KUKA KRL program: f1_Kuka_APT218T03S18.SRC

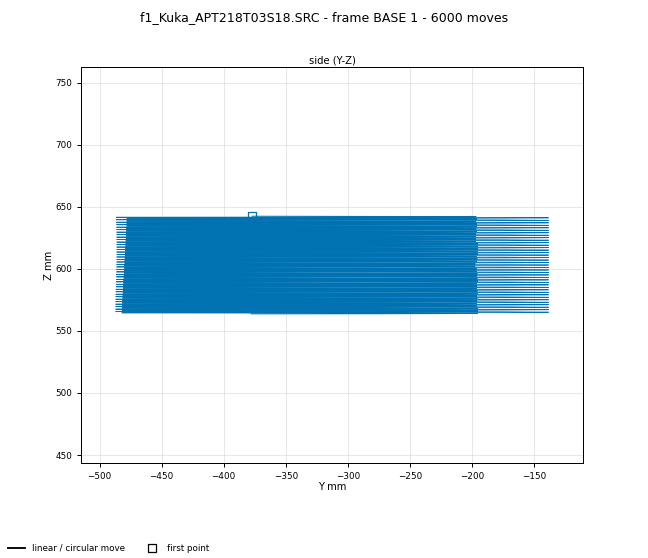
[picture p0: tool path of f1_Kuka_APT218T03S18.SRC in frame BASE 1, 6000 of 6001 moves have a stored position in this frame; points joined in program order, loops and branches not executed]
&ACCESS RVP
&REL 2
&PARAM TEMPLATE = C:\KRC\Roboter\Template\vorgabe
&PARAM EDITMASK = *
DEF f1_Kuka_APT218T03S18()


;FOLD INI;%{PE}%V3.2.0,%MKUKATPBASIS,%CINIT,%VCOMMON,%P
  ;FOLD BAS INI;%{E}%V3.2.0,%MKUKATPBASIS,%CINIT,%VINIT,%P
    GLOBAL INTERRUPT DECL 3 WHEN $STOPMESS==TRUE DO IR_STOPM ( )
    INTERRUPT ON 3
    BAS (#INITMOV,0 )
  ;ENDFOLD (BAS INI)
  ;FOLD USER INI;%{E}%V3.2.0,%MKUKATPUSER,%CINIT,%VINIT,%P
    ;Make your modifications here
  ;ENDFOLD (USER INI)
;ENDFOLD (INI)


;*** Make Null PTP Move
  PTP $pos_act

;*** Auto Load The Correct TOOL Data
  $tool=tool_data[3]

;*** Auto Load The Correct BASE Data
  $base=base_data[1]

  $ADVANCE = 5

;*** Restate Last Velocity
MMPM(30000.0)
SetRPM(6000)
LIN {X -0.101,Y -377.217,Z 642.442,A 0.000,B 0.000,C 90.000,E1 79.634} C_DIS
LIN {X 0.001,Y -366.007,Z 642.429,A 0.000,B 0.000,C 90.000,E1 77.285} C_DIS
LIN {X 0.196,Y -351.281,Z 642.411,A 0.000,B 0.000,C 90.000,E1 73.976} C_DIS
LIN {X -0.048,Y -341.253,Z 642.398,A 0.000,B 0.000,C 90.000,E1 71.583} C_DIS
LIN {X 0.012,Y -327.143,Z 642.377,A 0.000,B 0.000,C 90.000,E1 67.847} C_DIS
LIN {X 0.084,Y -314.471,Z 642.356,A 0.000,B 0.000,C 90.000,E1 64.024} C_DIS
LIN {X 0.048,Y -304.930,Z 642.338,A 0.000,B 0.000,C 90.000,E1 60.795} C_DIS
LIN {X -0.099,Y -296.125,Z 642.320,A 0.000,B 0.000,C 90.000,E1 57.533} C_DIS
LIN {X -0.021,Y -289.495,Z 642.305,A 0.000,B 0.000,C 90.000,E1 54.848} C_DIS
LIN {X -0.014,Y -283.083,Z 642.290,A 0.000,B 0.000,C 90.000,E1 52.145} C_DIS
LIN {X 0.119,Y -278.142,Z 642.278,A 0.000,B 0.000,C 90.000,E1 50.070} C_DIS
LIN {X 0.131,Y -272.810,Z 642.267,A 0.000,B 0.000,C 90.000,E1 48.000} C_DIS
LIN {X -0.152,Y -266.946,Z 642.255,A 0.000,B 0.000,C 90.000,E1 45.972} C_DIS
LIN {X -0.168,Y -260.527,Z 642.243,A 0.000,B 0.000,C 90.000,E1 43.866} C_DIS
LIN {X 0.065,Y -253.879,Z 642.232,A 0.000,B 0.000,C 90.000,E1 41.676} C_DIS
LIN {X -0.149,Y -243.020,Z 642.211,A 0.000,B 0.000,C 90.000,E1 38.096} C_DIS
LIN {X -0.001,Y -234.963,Z 642.195,A 0.000,B 0.000,C 90.000,E1 35.105} C_DIS
LIN {X 0.062,Y -227.705,Z 642.178,A 0.000,B 0.000,C 90.000,E1 32.084} C_DIS
LIN {X -0.103,Y -221.117,Z 642.161,A 0.000,B 0.000,C 90.000,E1 29.077} C_DIS
LIN {X -0.063,Y -215.336,Z 642.144,A 0.000,B 0.000,C 90.000,E1 25.976} C_DIS
LIN {X 0.066,Y -209.174,Z 642.122,A 0.000,B 0.000,C 90.000,E1 22.025} C_DIS
LIN {X 0.077,Y -204.198,Z 642.100,A 0.000,B 0.000,C 90.000,E1 18.055} C_DIS
LIN {X 0.016,Y -200.306,Z 642.078,A 0.000,B 0.000,C 90.000,E1 14.064} C_DIS
LIN {X 0.027,Y -196.658,Z 642.047,A 0.000,B 0.000,C 90.000,E1 8.398} C_DIS
LIN {X -0.004,Y -197.458,Z 641.952,A 0.000,B 0.000,C 90.000,E1 351.376} C_DIS
LIN {X -0.032,Y -200.895,Z 641.925,A 0.000,B 0.000,C 90.000,E1 346.520} C_DIS
LIN {X -0.002,Y -204.863,Z 641.903,A 0.000,B 0.000,C 90.000,E1 342.489} C_DIS
LIN {X -0.060,Y -209.769,Z 641.881,A 0.000,B 0.000,C 90.000,E1 338.518} C_DIS
LIN {X 0.082,Y -215.497,Z 641.859,A 0.000,B 0.000,C 90.000,E1 334.537} C_DIS
LIN {X -0.009,Y -221.886,Z 641.837,A 0.000,B 0.000,C 90.000,E1 330.667} C_DIS
LIN {X 0.024,Y -227.475,Z 641.820,A 0.000,B 0.000,C 90.000,E1 327.582} C_DIS
LIN {X 0.036,Y -234.865,Z 641.799,A 0.000,B 0.000,C 90.000,E1 323.783} C_DIS
LIN {X -0.064,Y -242.913,Z 641.778,A 0.000,B 0.000,C 90.000,E1 320.070} C_DIS
LIN {X 0.005,Y -251.812,Z 641.758,A 0.000,B 0.000,C 90.000,E1 316.377} C_DIS
LIN {X -0.006,Y -261.731,Z 641.738,A 0.000,B 0.000,C 90.000,E1 312.771} C_DIS
LIN {X 0.117,Y -271.858,Z 641.720,A 0.000,B 0.000,C 90.000,E1 309.564} C_DIS
LIN {X 0.057,Y -283.236,Z 641.703,A 0.000,B 0.000,C 90.000,E1 306.457} C_DIS
LIN {X -0.012,Y -295.817,Z 641.686,A 0.000,B 0.000,C 90.000,E1 303.420} C_DIS
LIN {X -0.138,Y -309.656,Z 641.669,A 0.000,B 0.000,C 90.000,E1 300.463} C_DIS
LIN {X 0.023,Y -323.063,Z 641.655,A 0.000,B 0.000,C 90.000,E1 297.847} C_DIS
LIN {X -0.032,Y -335.104,Z 641.642,A 0.000,B 0.000,C 90.000,E1 295.643} C_DIS
LIN {X 0.079,Y -351.402,Z 641.627,A 0.000,B 0.000,C 90.000,E1 292.845} C_DIS
LIN {X -0.048,Y -370.901,Z 641.610,A 0.000,B 0.000,C 90.000,E1 289.866} C_DIS
LIN {X -0.020,Y -386.121,Z 641.599,A 0.000,B 0.000,C 90.000,E1 287.819} C_DIS
LIN {X -0.151,Y -402.387,Z 641.588,A 0.000,B 0.000,C 90.000,E1 285.843} C_DIS
LIN {X 0.020,Y -414.001,Z 641.580,A 0.000,B 0.000,C 90.000,E1 284.426} C_DIS
LIN {X -0.039,Y -425.082,Z 641.573,A 0.000,B 0.000,C 90.000,E1 283.063} C_DIS
LIN {X -0.027,Y -435.735,Z 641.565,A 0.000,B 0.000,C 90.000,E1 281.715} C_DIS
LIN {X -0.081,Y -443.889,Z 641.559,A 0.000,B 0.000,C 90.000,E1 280.658} C_DIS
LIN {X -0.145,Y -456.034,Z 641.550,A 0.000,B 0.000,C 90.000,E1 279.095} C_DIS
LIN {X -0.043,Y -464.453,Z 641.545,A 0.000,B 0.000,C 90.000,E1 278.049} C_DIS
LIN {X -0.153,Y -470.095,Z 641.540,A 0.000,B 0.000,C 90.000,E1 277.296} C_DIS
LIN {X 0.259,Y -474.932,Z 641.536,A 0.000,B 0.000,C 90.000,E1 276.486} C_DIS
LIN {X 0.187,Y -478.977,Z 641.532,A 0.000,B 0.000,C 90.000,E1 275.739} C_DIS
LIN {X -0.142,Y -481.189,Z 641.529,A 0.000,B 0.000,C 90.000,E1 275.277} C_DIS
LIN {X 0.019,Y -482.986,Z 641.526,A 0.000,B 0.000,C 90.000,E1 274.759} C_DIS
LIN {X 0.149,Y -484.460,Z 641.524,A 0.000,B 0.000,C 90.000,E1 274.245} C_DIS
LIN {X -0.157,Y -485.468,Z 641.521,A 0.000,B 0.000,C 90.000,E1 273.784} C_DIS
LIN {X -0.002,Y -486.133,Z 641.518,A 0.000,B 0.000,C 90.000,E1 273.269} C_DIS
LIN {X 0.187,Y -486.492,Z 641.515,A 0.000,B 0.000,C 90.000,E1 272.751} C_DIS
LIN {X -0.130,Y -486.583,Z 641.513,A 0.000,B 0.000,C 90.000,E1 272.293} C_DIS
LIN {X 0.058,Y -486.383,Z 641.510,A 0.000,B 0.000,C 90.000,E1 271.776} C_DIS
LIN {X 0.230,Y -485.845,Z 641.507,A 0.000,B 0.000,C 90.000,E1 271.260} C_DIS
LIN {X -0.083,Y -484.907,Z 641.504,A 0.000,B 0.000,C 90.000,E1 270.802} C_DIS
LIN {X 0.088,Y -483.494,Z 641.502,A 0.000,B 0.000,C 90.000,E1 270.286} C_DIS
LIN {X -0.230,Y -481.516,Z 641.499,A 0.000,B 0.000,C 90.000,E1 269.828} C_DIS
LIN {X -0.074,Y -478.834,Z 641.496,A 0.000,B 0.000,C 90.000,E1 269.312} C_DIS
LIN {X 0.061,Y -475.404,Z 641.493,A 0.000,B 0.000,C 90.000,E1 268.797} C_DIS
LIN {X 0.175,Y -470.957,Z 641.491,A 0.000,B 0.000,C 90.000,E1 268.282} C_DIS
LIN {X 0.002,Y -468.333,Z 641.489,A 0.000,B 0.000,C 90.000,E1 268.051} C_DIS
LIN {X -0.184,Y -465.346,Z 641.488,A 0.000,B 0.000,C 90.000,E1 267.822} C_DIS
LIN {X -0.130,Y -462.383,Z 641.487,A 0.000,B 0.000,C 90.000,E1 267.593} C_DIS
LIN {X -0.076,Y -459.035,Z 641.485,A 0.000,B 0.000,C 90.000,E1 267.364} C_DIS
LIN {X 0.127,Y -452.068,Z 641.483,A 0.000,B 0.000,C 90.000,E1 266.963} C_DIS
LIN {X 0.044,Y -444.600,Z 641.482,A 0.000,B 0.000,C 90.000,E1 266.674} C_DIS
LIN {X 0.025,Y -436.739,Z 641.480,A 0.000,B 0.000,C 90.000,E1 266.445} C_DIS
LIN {X 0.024,Y -427.995,Z 641.479,A 0.000,B 0.000,C 90.000,E1 266.274} C_DIS
LIN {X -0.186,Y -419.938,Z 641.479,A 0.000,B 0.000,C 90.000,E1 266.216} C_DIS
LIN {X -0.026,Y -411.170,Z 641.479,A 0.000,B 0.000,C 90.000,E1 266.159} C_DIS
LIN {X -0.034,Y -180.927,Z 641.479,A 0.000,B 0.000,C 90.000,E1 266.159} C_DIS
LIN {X 0.072,Y -180.902,Z 641.474,A 0.000,B 0.000,C 90.000,E1 265.241} C_DIS
LIN {X 0.021,Y -180.228,Z 641.464,A 0.000,B 0.000,C 90.000,E1 263.571} C_DIS
LIN {X -0.025,Y -179.041,Z 641.446,A 0.000,B 0.000,C 90.000,E1 260.208} C_DIS
LIN {X 0.037,Y -178.709,Z 641.441,A 0.000,B 0.000,C 90.000,E1 259.342} C_DIS
LIN {X -0.069,Y -175.758,Z 641.413,A 0.000,B 0.000,C 90.000,E1 254.283} C_DIS
LIN {X -0.019,Y -171.942,Z 641.384,A 0.000,B 0.000,C 90.000,E1 249.135} C_DIS
LIN {X -0.044,Y -171.326,Z 641.379,A 0.000,B 0.000,C 90.000,E1 248.284} C_DIS
LIN {X 0.010,Y -167.582,Z 641.355,A 0.000,B 0.000,C 90.000,E1 243.948} C_DIS
LIN {X -0.052,Y -166.217,Z 641.346,A 0.000,B 0.000,C 90.000,E1 242.231} C_DIS
LIN {X -0.063,Y -162.980,Z 641.326,A 0.000,B 0.000,C 90.000,E1 238.742} C_DIS
LIN {X -0.015,Y -160.894,Z 641.312,A 0.000,B 0.000,C 90.000,E1 236.087} C_DIS
LIN {X -0.038,Y -157.663,Z 641.292,A 0.000,B 0.000,C 90.000,E1 232.557} C_DIS
LIN {X -0.099,Y -155.701,Z 641.277,A 0.000,B 0.000,C 90.000,E1 229.908} C_DIS
LIN {X -0.044,Y -151.964,Z 641.252,A 0.000,B 0.000,C 90.000,E1 225.405} C_DIS
LIN {X -0.027,Y -150.205,Z 641.237,A 0.000,B 0.000,C 90.000,E1 222.690} C_DIS
LIN {X -0.012,Y -146.973,Z 641.212,A 0.000,B 0.000,C 90.000,E1 218.141} C_DIS
LIN {X 0.007,Y -145.560,Z 641.197,A 0.000,B 0.000,C 90.000,E1 215.391} C_DIS
LIN {X 0.006,Y -142.952,Z 641.171,A 0.000,B 0.000,C 90.000,E1 210.797} C_DIS
LIN {X -0.063,Y -141.577,Z 641.151,A 0.000,B 0.000,C 90.000,E1 207.129} C_DIS
LIN {X -0.016,Y -139.415,Z 641.114,A 0.000,B 0.000,C 90.000,E1 200.610} C_DIS
LIN {X 0.037,Y -139.139,Z 641.104,A 0.000,B 0.000,C 90.000,E1 198.725} C_DIS
LIN {X 0.063,Y -138.348,Z 641.057,A 0.000,B 0.000,C 90.000,E1 190.310} C_DIS
LIN {X 0.051,Y -139.493,Z 641.006,A 0.000,B 0.000,C 90.000,E1 180.974} C_DIS
LIN {X -0.008,Y -141.105,Z 640.974,A 0.000,B 0.000,C 90.000,E1 175.412} C_DIS
LIN {X -0.055,Y -142.484,Z 640.959,A 0.000,B 0.000,C 90.000,E1 172.648} C_DIS
LIN {X 0.034,Y -144.734,Z 640.933,A 0.000,B 0.000,C 90.000,E1 167.993} C_DIS
LIN {X -0.015,Y -147.339,Z 640.913,A 0.000,B 0.000,C 90.000,E1 164.338} C_DIS
LIN {X 0.050,Y -150.663,Z 640.888,A 0.000,B 0.000,C 90.000,E1 159.752} C_DIS
LIN {X -0.070,Y -154.141,Z 640.867,A 0.000,B 0.000,C 90.000,E1 156.177} C_DIS
LIN {X -0.006,Y -157.570,Z 640.848,A 0.000,B 0.000,C 90.000,E1 152.564} C_DIS
LIN {X 0.018,Y -161.815,Z 640.828,A 0.000,B 0.000,C 90.000,E1 148.997} C_DIS
LIN {X 0.037,Y -166.006,Z 640.808,A 0.000,B 0.000,C 90.000,E1 145.468} C_DIS
LIN {X 0.029,Y -171.005,Z 640.789,A 0.000,B 0.000,C 90.000,E1 141.984} C_DIS
LIN {X -0.056,Y -175.875,Z 640.770,A 0.000,B 0.000,C 90.000,E1 138.566} C_DIS
LIN {X -0.062,Y -181.480,Z 640.751,A 0.000,B 0.000,C 90.000,E1 135.162} C_DIS
LIN {X 0.074,Y -186.993,Z 640.732,A 0.000,B 0.000,C 90.000,E1 131.757} C_DIS
LIN {X -0.127,Y -191.046,Z 640.720,A 0.000,B 0.000,C 90.000,E1 129.644} C_DIS
LIN {X 0.183,Y -288.245,Z 640.720,A 0.000,B 0.000,C 90.000,E1 129.564} C_DIS
LIN {X 0.022,Y -293.362,Z 640.719,A 0.000,B 0.000,C 90.000,E1 129.439} C_DIS
LIN {X 0.045,Y -295.630,Z 640.718,A 0.000,B 0.000,C 90.000,E1 129.277} C_DIS
LIN {X -0.029,Y -299.485,Z 640.716,A 0.000,B 0.000,C 90.000,E1 128.874} C_DIS
LIN {X 0.125,Y -301.412,Z 640.714,A 0.000,B 0.000,C 90.000,E1 128.543} C_DIS
LIN {X 0.045,Y -302.930,Z 640.713,A 0.000,B 0.000,C 90.000,E1 128.257} C_DIS
LIN {X 0.001,Y -304.249,Z 640.711,A 0.000,B 0.000,C 90.000,E1 127.935} C_DIS
LIN {X -0.007,Y -307.079,Z 640.705,A 0.000,B 0.000,C 90.000,E1 126.950} C_DIS
LIN {X -0.065,Y -316.926,Z 640.687,A 0.000,B 0.000,C 90.000,E1 123.706} C_DIS
LIN {X 0.125,Y -327.091,Z 640.671,A 0.000,B 0.000,C 90.000,E1 120.797} C_DIS
LIN {X 0.117,Y -338.594,Z 640.656,A 0.000,B 0.000,C 90.000,E1 117.975} C_DIS
LIN {X 0.123,Y -351.535,Z 640.640,A 0.000,B 0.000,C 90.000,E1 115.207} C_DIS
LIN {X -0.029,Y -364.342,Z 640.627,A 0.000,B 0.000,C 90.000,E1 112.823} C_DIS
LIN {X -0.149,Y -378.471,Z 640.614,A 0.000,B 0.000,C 90.000,E1 110.482} C_DIS
LIN {X -0.180,Y -394.024,Z 640.601,A 0.000,B 0.000,C 90.000,E1 108.181} C_DIS
LIN {X 0.061,Y -411.113,Z 640.588,A 0.000,B 0.000,C 90.000,E1 105.898} C_DIS
LIN {X 0.004,Y -429.864,Z 640.576,A 0.000,B 0.000,C 90.000,E1 103.716} C_DIS
LIN {X -0.128,Y -449.867,Z 640.565,A 0.000,B 0.000,C 90.000,E1 101.658} C_DIS
LIN {X 0.105,Y -470.432,Z 640.554,A 0.000,B 0.000,C 90.000,E1 99.726} C_DIS
LIN {X 0.090,Y -472.590,Z 640.553,A 0.000,B 0.000,C 90.000,E1 99.500} C_DIS
LIN {X -0.055,Y -474.386,Z 640.551,A 0.000,B 0.000,C 90.000,E1 99.265} C_DIS
LIN {X -0.202,Y -475.734,Z 640.550,A 0.000,B 0.000,C 90.000,E1 99.029} C_DIS
LIN {X -0.078,Y -477.424,Z 640.547,A 0.000,B 0.000,C 90.000,E1 98.511} C_DIS
LIN {X 0.057,Y -478.042,Z 640.544,A 0.000,B 0.000,C 90.000,E1 97.992} C_DIS
LIN {X 0.205,Y -477.692,Z 640.542,A 0.000,B 0.000,C 90.000,E1 97.473} C_DIS
LIN {X -0.059,Y -476.322,Z 640.539,A 0.000,B 0.000,C 90.000,E1 97.004} C_DIS
LIN {X 0.223,Y -475.185,Z 640.537,A 0.000,B 0.000,C 90.000,E1 96.720} C_DIS
LIN {X 0.087,Y -473.668,Z 640.536,A 0.000,B 0.000,C 90.000,E1 96.486} C_DIS
LIN {X 0.027,Y -456.397,Z 640.522,A 0.000,B 0.000,C 90.000,E1 93.955} C_DIS
LIN {X -0.053,Y -444.173,Z 640.510,A 0.000,B 0.000,C 90.000,E1 91.892} C_DIS
LIN {X -0.121,Y -434.157,Z 640.500,A 0.000,B 0.000,C 90.000,E1 90.057} C_DIS
LIN {X 0.193,Y -426.734,Z 640.493,A 0.000,B 0.000,C 90.000,E1 88.682} C_DIS
LIN {X 0.085,Y -417.419,Z 640.484,A 0.000,B 0.000,C 90.000,E1 87.078} C_DIS
LIN {X 0.008,Y -404.942,Z 640.472,A 0.000,B 0.000,C 90.000,E1 84.894} C_DIS
LIN {X -0.190,Y -388.323,Z 640.454,A 0.000,B 0.000,C 90.000,E1 81.837} C_DIS
LIN {X 0.066,Y -374.000,Z 640.439,A 0.000,B 0.000,C 90.000,E1 78.926} C_DIS
LIN {X 0.011,Y -362.875,Z 640.425,A 0.000,B 0.000,C 90.000,E1 76.589} C_DIS
LIN {X -0.130,Y -347.171,Z 640.406,A 0.000,B 0.000,C 90.000,E1 73.015} C_DIS
LIN {X -0.047,Y -334.905,Z 640.388,A 0.000,B 0.000,C 90.000,E1 69.934} C_DIS
LIN {X -0.039,Y -322.527,Z 640.369,A 0.000,B 0.000,C 90.000,E1 66.485} C_DIS
LIN {X 0.175,Y -312.330,Z 640.352,A 0.000,B 0.000,C 90.000,E1 63.256} C_DIS
LIN {X -0.047,Y -302.974,Z 640.334,A 0.000,B 0.000,C 90.000,E1 60.049} C_DIS
LIN {X -0.085,Y -294.318,Z 640.315,A 0.000,B 0.000,C 90.000,E1 56.755} C_DIS
LIN {X -0.047,Y -287.750,Z 640.300,A 0.000,B 0.000,C 90.000,E1 54.069} C_DIS
LIN {X 0.003,Y -282.993,Z 640.289,A 0.000,B 0.000,C 90.000,E1 52.029} C_DIS
LIN {X -0.034,Y -278.021,Z 640.278,A 0.000,B 0.000,C 90.000,E1 49.989} C_DIS
LIN {X -0.015,Y -274.511,Z 640.270,A 0.000,B 0.000,C 90.000,E1 48.609} C_DIS
LIN {X -0.067,Y -268.817,Z 640.258,A 0.000,B 0.000,C 90.000,E1 46.539} C_DIS
LIN {X 0.017,Y -264.672,Z 640.251,A 0.000,B 0.000,C 90.000,E1 45.121} C_DIS
LIN {X -0.042,Y -258.115,Z 640.239,A 0.000,B 0.000,C 90.000,E1 43.014} C_DIS
LIN {X -0.015,Y -250.270,Z 640.225,A 0.000,B 0.000,C 90.000,E1 40.496} C_DIS
LIN {X -0.120,Y -240.741,Z 640.207,A 0.000,B 0.000,C 90.000,E1 37.237} C_DIS
LIN {X -0.033,Y -232.883,Z 640.190,A 0.000,B 0.000,C 90.000,E1 34.246} C_DIS
LIN {X 0.044,Y -225.831,Z 640.173,A 0.000,B 0.000,C 90.000,E1 31.209} C_DIS
LIN {X 0.023,Y -219.459,Z 640.156,A 0.000,B 0.000,C 90.000,E1 28.153} C_DIS
LIN {X -0.082,Y -213.910,Z 640.139,A 0.000,B 0.000,C 90.000,E1 25.079} C_DIS
LIN {X 0.110,Y -208.007,Z 640.117,A 0.000,B 0.000,C 90.000,E1 21.099} C_DIS
LIN {X 0.016,Y -203.310,Z 640.095,A 0.000,B 0.000,C 90.000,E1 17.149} C_DIS
LIN {X 0.068,Y -199.659,Z 640.073,A 0.000,B 0.000,C 90.000,E1 13.119} C_DIS
LIN {X 0.009,Y -196.320,Z 640.042,A 0.000,B 0.000,C 90.000,E1 7.466} C_DIS
LIN {X 0.013,Y -197.092,Z 639.957,A 0.000,B 0.000,C 90.000,E1 352.186} C_DIS
LIN {X -0.112,Y -200.285,Z 639.930,A 0.000,B 0.000,C 90.000,E1 347.353} C_DIS
LIN {X -0.108,Y -204.072,Z 639.907,A 0.000,B 0.000,C 90.000,E1 343.323} C_DIS
LIN {X -0.065,Y -208.785,Z 639.885,A 0.000,B 0.000,C 90.000,E1 339.316} C_DIS
LIN {X -0.037,Y -214.338,Z 639.863,A 0.000,B 0.000,C 90.000,E1 335.357} C_DIS
LIN {X 0.032,Y -220.591,Z 639.841,A 0.000,B 0.000,C 90.000,E1 331.435} C_DIS
LIN {X 0.042,Y -227.497,Z 639.820,A 0.000,B 0.000,C 90.000,E1 327.582} C_DIS
LIN {X 0.056,Y -234.883,Z 639.799,A 0.000,B 0.000,C 90.000,E1 323.783} C_DIS
LIN {X -0.045,Y -242.908,Z 639.778,A 0.000,B 0.000,C 90.000,E1 320.070} C_DIS
LIN {X 0.025,Y -251.767,Z 639.758,A 0.000,B 0.000,C 90.000,E1 316.377} C_DIS
LIN {X 0.014,Y -261.699,Z 639.738,A 0.000,B 0.000,C 90.000,E1 312.771} C_DIS
LIN {X 0.137,Y -271.799,Z 639.720,A 0.000,B 0.000,C 90.000,E1 309.564} C_DIS
LIN {X 0.076,Y -283.135,Z 639.703,A 0.000,B 0.000,C 90.000,E1 306.457} C_DIS
LIN {X 0.005,Y -295.730,Z 639.686,A 0.000,B 0.000,C 90.000,E1 303.420} C_DIS
LIN {X -0.123,Y -309.574,Z 639.669,A 0.000,B 0.000,C 90.000,E1 300.463} C_DIS
LIN {X 0.036,Y -322.972,Z 639.655,A 0.000,B 0.000,C 90.000,E1 297.847} C_DIS
LIN {X -0.021,Y -335.011,Z 639.642,A 0.000,B 0.000,C 90.000,E1 295.643} C_DIS
LIN {X 0.089,Y -351.302,Z 639.627,A 0.000,B 0.000,C 90.000,E1 292.845} C_DIS
LIN {X -0.041,Y -370.854,Z 639.610,A 0.000,B 0.000,C 90.000,E1 289.866} C_DIS
LIN {X -0.014,Y -386.061,Z 639.599,A 0.000,B 0.000,C 90.000,E1 287.819} C_DIS
LIN {X -0.145,Y -402.327,Z 639.588,A 0.000,B 0.000,C 90.000,E1 285.843} C_DIS
LIN {X 0.052,Y -413.886,Z 639.580,A 0.000,B 0.000,C 90.000,E1 284.426} C_DIS
LIN {X 0.019,Y -424.953,Z 639.573,A 0.000,B 0.000,C 90.000,E1 283.063} C_DIS
LIN {X 0.030,Y -435.614,Z 639.565,A 0.000,B 0.000,C 90.000,E1 281.715} C_DIS
LIN {X 0.193,Y -445.780,Z 639.558,A 0.000,B 0.000,C 90.000,E1 280.366} C_DIS
LIN {X 0.015,Y -464.248,Z 639.545,A 0.000,B 0.000,C 90.000,E1 278.049} C_DIS
LIN {X -0.096,Y -469.883,Z 639.540,A 0.000,B 0.000,C 90.000,E1 277.296} C_DIS
LIN {X -0.158,Y -474.781,Z 639.536,A 0.000,B 0.000,C 90.000,E1 276.543} C_DIS
LIN {X 0.240,Y -478.856,Z 639.532,A 0.000,B 0.000,C 90.000,E1 275.739} C_DIS
LIN {X -0.090,Y -481.064,Z 639.529,A 0.000,B 0.000,C 90.000,E1 275.277} C_DIS
LIN {X 0.071,Y -482.854,Z 639.526,A 0.000,B 0.000,C 90.000,E1 274.759} C_DIS
LIN {X 0.200,Y -484.296,Z 639.524,A 0.000,B 0.000,C 90.000,E1 274.245} C_DIS
LIN {X -0.106,Y -485.341,Z 639.521,A 0.000,B 0.000,C 90.000,E1 273.784} C_DIS
LIN {X 0.048,Y -486.015,Z 639.518,A 0.000,B 0.000,C 90.000,E1 273.269} C_DIS
LIN {X 0.236,Y -486.392,Z 639.515,A 0.000,B 0.000,C 90.000,E1 272.751} C_DIS
LIN {X -0.082,Y -486.504,Z 639.513,A 0.000,B 0.000,C 90.000,E1 272.293} C_DIS
LIN {X 0.106,Y -486.301,Z 639.510,A 0.000,B 0.000,C 90.000,E1 271.776} C_DIS
LIN {X -0.208,Y -485.820,Z 639.507,A 0.000,B 0.000,C 90.000,E1 271.318} C_DIS
LIN {X -0.036,Y -484.879,Z 639.504,A 0.000,B 0.000,C 90.000,E1 270.802} C_DIS
LIN {X 0.134,Y -483.461,Z 639.502,A 0.000,B 0.000,C 90.000,E1 270.286} C_DIS
LIN {X -0.185,Y -481.479,Z 639.499,A 0.000,B 0.000,C 90.000,E1 269.828} C_DIS
LIN {X -0.028,Y -478.866,Z 639.496,A 0.000,B 0.000,C 90.000,E1 269.312} C_DIS
LIN {X 0.107,Y -475.448,Z 639.493,A 0.000,B 0.000,C 90.000,E1 268.797} C_DIS
LIN {X 0.221,Y -471.036,Z 639.491,A 0.000,B 0.000,C 90.000,E1 268.282} C_DIS
LIN {X 0.047,Y -468.418,Z 639.489,A 0.000,B 0.000,C 90.000,E1 268.051} C_DIS
LIN {X -0.083,Y -462.497,Z 639.487,A 0.000,B 0.000,C 90.000,E1 267.593} C_DIS
LIN {X -0.027,Y -459.192,Z 639.485,A 0.000,B 0.000,C 90.000,E1 267.364} C_DIS
LIN {X -0.166,Y -455.931,Z 639.484,A 0.000,B 0.000,C 90.000,E1 267.192} C_DIS
LIN {X 0.148,Y -452.156,Z 639.483,A 0.000,B 0.000,C 90.000,E1 266.963} C_DIS
LIN {X 0.078,Y -444.735,Z 639.482,A 0.000,B 0.000,C 90.000,E1 266.674} C_DIS
LIN {X 0.060,Y -436.947,Z 639.480,A 0.000,B 0.000,C 90.000,E1 266.445} C_DIS
LIN {X 0.058,Y -428.482,Z 639.479,A 0.000,B 0.000,C 90.000,E1 266.274} C_DIS
LIN {X -0.169,Y -420.878,Z 639.479,A 0.000,B 0.000,C 90.000,E1 266.216} C_DIS
LIN {X -0.019,Y -413.648,Z 639.479,A 0.000,B 0.000,C 90.000,E1 266.159} C_DIS
LIN {X -0.032,Y -180.926,Z 639.479,A 0.000,B 0.000,C 90.000,E1 266.159} C_DIS
LIN {X 0.065,Y -180.901,Z 639.474,A 0.000,B 0.000,C 90.000,E1 265.241} C_DIS
LIN {X 0.015,Y -180.227,Z 639.464,A 0.000,B 0.000,C 90.000,E1 263.571} C_DIS
LIN {X -0.032,Y -179.040,Z 639.446,A 0.000,B 0.000,C 90.000,E1 260.208} C_DIS
LIN {X 0.030,Y -178.709,Z 639.441,A 0.000,B 0.000,C 90.000,E1 259.342} C_DIS
LIN {X -0.029,Y -175.757,Z 639.413,A 0.000,B 0.000,C 90.000,E1 254.267} C_DIS
LIN {X -0.026,Y -171.940,Z 639.384,A 0.000,B 0.000,C 90.000,E1 249.135} C_DIS
LIN {X -0.050,Y -171.324,Z 639.379,A 0.000,B 0.000,C 90.000,E1 248.284} C_DIS
LIN {X 0.002,Y -167.580,Z 639.355,A 0.000,B 0.000,C 90.000,E1 243.948} C_DIS
LIN {X -0.058,Y -166.215,Z 639.346,A 0.000,B 0.000,C 90.000,E1 242.231} C_DIS
LIN {X -0.069,Y -162.977,Z 639.326,A 0.000,B 0.000,C 90.000,E1 238.742} C_DIS
LIN {X -0.022,Y -160.892,Z 639.312,A 0.000,B 0.000,C 90.000,E1 236.087} C_DIS
LIN {X -0.044,Y -157.661,Z 639.292,A 0.000,B 0.000,C 90.000,E1 232.557} C_DIS
LIN {X 0.013,Y -155.699,Z 639.277,A 0.000,B 0.000,C 90.000,E1 229.865} C_DIS
LIN {X -0.050,Y -151.963,Z 639.252,A 0.000,B 0.000,C 90.000,E1 225.405} C_DIS
LIN {X -0.033,Y -150.203,Z 639.237,A 0.000,B 0.000,C 90.000,E1 222.690} C_DIS
LIN {X -0.018,Y -146.972,Z 639.212,A 0.000,B 0.000,C 90.000,E1 218.141} C_DIS
LIN {X 0.000,Y -145.559,Z 639.197,A 0.000,B 0.000,C 90.000,E1 215.391} C_DIS
LIN {X 0.000,Y -142.951,Z 639.171,A 0.000,B 0.000,C 90.000,E1 210.797} C_DIS
LIN {X -0.069,Y -141.576,Z 639.151,A 0.000,B 0.000,C 90.000,E1 207.129} C_DIS
LIN {X -0.021,Y -139.414,Z 639.114,A 0.000,B 0.000,C 90.000,E1 200.610} C_DIS
LIN {X 0.031,Y -139.138,Z 639.104,A 0.000,B 0.000,C 90.000,E1 198.725} C_DIS
LIN {X 0.057,Y -138.348,Z 639.057,A 0.000,B 0.000,C 90.000,E1 190.310} C_DIS
LIN {X 0.046,Y -139.493,Z 639.005,A 0.000,B 0.000,C 90.000,E1 180.974} C_DIS
LIN {X -0.014,Y -141.106,Z 638.974,A 0.000,B 0.000,C 90.000,E1 175.412} C_DIS
LIN {X -0.060,Y -142.485,Z 638.959,A 0.000,B 0.000,C 90.000,E1 172.648} C_DIS
LIN {X 0.028,Y -144.735,Z 638.933,A 0.000,B 0.000,C 90.000,E1 167.993} C_DIS
LIN {X -0.021,Y -147.340,Z 638.913,A 0.000,B 0.000,C 90.000,E1 164.338} C_DIS
LIN {X 0.043,Y -150.664,Z 638.888,A 0.000,B 0.000,C 90.000,E1 159.752} C_DIS
LIN {X -0.075,Y -154.144,Z 638.867,A 0.000,B 0.000,C 90.000,E1 156.177} C_DIS
LIN {X 0.059,Y -157.573,Z 638.848,A 0.000,B 0.000,C 90.000,E1 152.538} C_DIS
LIN {X 0.011,Y -161.818,Z 638.828,A 0.000,B 0.000,C 90.000,E1 148.997} C_DIS
LIN {X 0.029,Y -166.009,Z 638.808,A 0.000,B 0.000,C 90.000,E1 145.468} C_DIS
LIN {X 0.022,Y -171.008,Z 638.789,A 0.000,B 0.000,C 90.000,E1 141.984} C_DIS
LIN {X 0.054,Y -175.878,Z 638.770,A 0.000,B 0.000,C 90.000,E1 138.528} C_DIS
LIN {X -0.070,Y -181.483,Z 638.751,A 0.000,B 0.000,C 90.000,E1 135.162} C_DIS
LIN {X 0.066,Y -186.997,Z 638.732,A 0.000,B 0.000,C 90.000,E1 131.757} C_DIS
LIN {X 0.113,Y -191.060,Z 638.720,A 0.000,B 0.000,C 90.000,E1 129.564} C_DIS
LIN {X 0.119,Y -288.917,Z 638.720,A 0.000,B 0.000,C 90.000,E1 129.564} C_DIS
LIN {X -0.039,Y -290.500,Z 638.720,A 0.000,B 0.000,C 90.000,E1 129.564} C_DIS
LIN {X 0.033,Y -295.571,Z 638.718,A 0.000,B 0.000,C 90.000,E1 129.277} C_DIS
LIN {X -0.012,Y -298.795,Z 638.716,A 0.000,B 0.000,C 90.000,E1 128.955} C_DIS
LIN {X -0.049,Y -302.392,Z 638.713,A 0.000,B 0.000,C 90.000,E1 128.382} C_DIS
LIN {X 0.136,Y -303.831,Z 638.711,A 0.000,B 0.000,C 90.000,E1 128.016} C_DIS
LIN {X -0.104,Y -304.963,Z 638.709,A 0.000,B 0.000,C 90.000,E1 127.729} C_DIS
LIN {X -0.001,Y -315.525,Z 638.690,A 0.000,B 0.000,C 90.000,E1 124.119} C_DIS
LIN {X -0.129,Y -325.503,Z 638.674,A 0.000,B 0.000,C 90.000,E1 121.258} C_DIS
LIN {X -0.030,Y -336.801,Z 638.658,A 0.000,B 0.000,C 90.000,E1 118.409} C_DIS
LIN {X -0.093,Y -349.529,Z 638.642,A 0.000,B 0.000,C 90.000,E1 115.643} C_DIS
LIN {X 0.027,Y -362.127,Z 638.629,A 0.000,B 0.000,C 90.000,E1 113.206} C_DIS
LIN {X -0.006,Y -376.032,Z 638.616,A 0.000,B 0.000,C 90.000,E1 110.844} C_DIS
LIN {X -0.097,Y -391.343,Z 638.603,A 0.000,B 0.000,C 90.000,E1 108.544} C_DIS
LIN {X 0.081,Y -408.173,Z 638.590,A 0.000,B 0.000,C 90.000,E1 106.260} C_DIS
LIN {X 0.059,Y -426.642,Z 638.578,A 0.000,B 0.000,C 90.000,E1 104.064} C_DIS
LIN {X 0.146,Y -446.524,Z 638.566,A 0.000,B 0.000,C 90.000,E1 101.951} C_DIS
LIN {X 0.170,Y -467.009,Z 638.556,A 0.000,B 0.000,C 90.000,E1 100.018} C_DIS
LIN {X 0.207,Y -471.980,Z 638.553,A 0.000,B 0.000,C 90.000,E1 99.557} C_DIS
LIN {X 0.164,Y -473.868,Z 638.552,A 0.000,B 0.000,C 90.000,E1 99.321} C_DIS
LIN {X 0.045,Y -475.304,Z 638.551,A 0.000,B 0.000,C 90.000,E1 99.095} C_DIS
LIN {X 0.242,Y -477.252,Z 638.548,A 0.000,B 0.000,C 90.000,E1 98.568} C_DIS
LIN {X -0.099,Y -478.081,Z 638.545,A 0.000,B 0.000,C 90.000,E1 98.106} C_DIS
LIN {X 0.047,Y -477.933,Z 638.542,A 0.000,B 0.000,C 90.000,E1 97.587} C_DIS
LIN {X 0.198,Y -476.789,Z 638.539,A 0.000,B 0.000,C 90.000,E1 97.068} C_DIS
LIN {X 0.064,Y -475.790,Z 638.538,A 0.000,B 0.000,C 90.000,E1 96.834} C_DIS
LIN {X -0.125,Y -474.444,Z 638.537,A 0.000,B 0.000,C 90.000,E1 96.606} C_DIS
LIN {X 0.121,Y -455.510,Z 638.521,A 0.000,B 0.000,C 90.000,E1 93.784} C_DIS
LIN {X 0.036,Y -443.364,Z 638.510,A 0.000,B 0.000,C 90.000,E1 91.718} C_DIS
LIN {X -0.058,Y -433.360,Z 638.499,A 0.000,B 0.000,C 90.000,E1 89.885} C_DIS
LIN {X -0.188,Y -425.913,Z 638.492,A 0.000,B 0.000,C 90.000,E1 88.568} C_DIS
LIN {X -0.179,Y -414.977,Z 638.481,A 0.000,B 0.000,C 90.000,E1 86.674} C_DIS
LIN {X 0.012,Y -404.073,Z 638.471,A 0.000,B 0.000,C 90.000,E1 84.723} C_DIS
LIN {X 0.170,Y -388.981,Z 638.455,A 0.000,B 0.000,C 90.000,E1 81.894} C_DIS
LIN {X -0.003,Y -374.651,Z 638.439,A 0.000,B 0.000,C 90.000,E1 79.050} C_DIS
LIN {X 0.035,Y -363.508,Z 638.426,A 0.000,B 0.000,C 90.000,E1 76.700} C_DIS
LIN {X -0.176,Y -347.771,Z 638.406,A 0.000,B 0.000,C 90.000,E1 73.142} C_DIS
LIN {X -0.070,Y -336.723,Z 638.391,A 0.000,B 0.000,C 90.000,E1 70.369} C_DIS
LIN {X -0.053,Y -323.098,Z 638.370,A 0.000,B 0.000,C 90.000,E1 66.613} C_DIS
LIN {X 0.149,Y -310.949,Z 638.349,A 0.000,B 0.000,C 90.000,E1 62.743} C_DIS
LIN {X -0.117,Y -301.713,Z 638.331,A 0.000,B 0.000,C 90.000,E1 59.537} C_DIS
LIN {X -0.042,Y -293.158,Z 638.312,A 0.000,B 0.000,C 90.000,E1 56.215} C_DIS
LIN {X 0.013,Y -285.042,Z 638.294,A 0.000,B 0.000,C 90.000,E1 52.844} C_DIS
LIN {X 0.012,Y -280.205,Z 638.282,A 0.000,B 0.000,C 90.000,E1 50.803} C_DIS
LIN {X -0.115,Y -275.056,Z 638.271,A 0.000,B 0.000,C 90.000,E1 48.771} C_DIS
LIN {X 0.028,Y -269.366,Z 638.259,A 0.000,B 0.000,C 90.000,E1 46.662} C_DIS
LIN {X 0.123,Y -265.255,Z 638.252,A 0.000,B 0.000,C 90.000,E1 45.243} C_DIS
LIN {X 0.067,Y -258.712,Z 638.240,A 0.000,B 0.000,C 90.000,E1 43.137} C_DIS
LIN {X 0.096,Y -250.840,Z 638.226,A 0.000,B 0.000,C 90.000,E1 40.620} C_DIS
LIN {X -0.005,Y -241.261,Z 638.208,A 0.000,B 0.000,C 90.000,E1 37.363} C_DIS
LIN {X -0.043,Y -233.386,Z 638.191,A 0.000,B 0.000,C 90.000,E1 34.405} C_DIS
LIN {X -0.024,Y -226.303,Z 638.174,A 0.000,B 0.000,C 90.000,E1 31.386} C_DIS
LIN {X 0.052,Y -219.895,Z 638.157,A 0.000,B 0.000,C 90.000,E1 28.309} C_DIS
LIN {X 0.058,Y -214.273,Z 638.140,A 0.000,B 0.000,C 90.000,E1 25.207} C_DIS
LIN {X 0.034,Y -209.427,Z 638.123,A 0.000,B 0.000,C 90.000,E1 22.078} C_DIS
LIN {X -0.015,Y -204.441,Z 638.101,A 0.000,B 0.000,C 90.000,E1 18.127} C_DIS
LIN {X -0.009,Y -200.509,Z 638.078,A 0.000,B 0.000,C 90.000,E1 14.120} C_DIS
LIN {X 0.008,Y -196.843,Z 638.047,A 0.000,B 0.000,C 90.000,E1 8.454} C_DIS
LIN {X 0.005,Y -197.602,Z 637.952,A 0.000,B 0.000,C 90.000,E1 351.376} C_DIS
LIN {X -0.017,Y -201.034,Z 637.925,A 0.000,B 0.000,C 90.000,E1 346.520} C_DIS
LIN {X 0.016,Y -205.013,Z 637.903,A 0.000,B 0.000,C 90.000,E1 342.489} C_DIS
LIN {X -0.037,Y -209.892,Z 637.881,A 0.000,B 0.000,C 90.000,E1 338.518} C_DIS
LIN {X -0.084,Y -215.605,Z 637.859,A 0.000,B 0.000,C 90.000,E1 334.588} C_DIS
LIN {X 0.023,Y -221.956,Z 637.837,A 0.000,B 0.000,C 90.000,E1 330.667} C_DIS
LIN {X -0.007,Y -228.965,Z 637.816,A 0.000,B 0.000,C 90.000,E1 326.834} C_DIS
LIN {X 0.074,Y -234.906,Z 637.799,A 0.000,B 0.000,C 90.000,E1 323.783} C_DIS
LIN {X -0.025,Y -242.902,Z 637.778,A 0.000,B 0.000,C 90.000,E1 320.070} C_DIS
LIN {X 0.045,Y -251.744,Z 637.758,A 0.000,B 0.000,C 90.000,E1 316.377} C_DIS
LIN {X 0.034,Y -261.651,Z 637.738,A 0.000,B 0.000,C 90.000,E1 312.771} C_DIS
LIN {X 0.156,Y -271.738,Z 637.720,A 0.000,B 0.000,C 90.000,E1 309.564} C_DIS
LIN {X 0.093,Y -283.040,Z 637.703,A 0.000,B 0.000,C 90.000,E1 306.457} C_DIS
LIN {X 0.013,Y -297.110,Z 637.684,A 0.000,B 0.000,C 90.000,E1 303.086} C_DIS
LIN {X -0.067,Y -311.121,Z 637.667,A 0.000,B 0.000,C 90.000,E1 300.129} C_DIS
LIN {X 0.050,Y -322.871,Z 637.655,A 0.000,B 0.000,C 90.000,E1 297.847} C_DIS
LIN {X -0.009,Y -334.897,Z 637.642,A 0.000,B 0.000,C 90.000,E1 295.643} C_DIS
LIN {X 0.080,Y -349.351,Z 637.629,A 0.000,B 0.000,C 90.000,E1 293.153} C_DIS
LIN {X -0.111,Y -368.736,Z 637.612,A 0.000,B 0.000,C 90.000,E1 290.174} C_DIS
LIN {X -0.138,Y -383.765,Z 637.601,A 0.000,B 0.000,C 90.000,E1 288.127} C_DIS
LIN {X -0.140,Y -402.268,Z 637.588,A 0.000,B 0.000,C 90.000,E1 285.843} C_DIS
LIN {X -0.082,Y -411.571,Z 637.582,A 0.000,B 0.000,C 90.000,E1 284.717} C_DIS
LIN {X -0.175,Y -422.743,Z 637.574,A 0.000,B 0.000,C 90.000,E1 283.355} C_DIS
LIN {X -0.210,Y -433.517,Z 637.567,A 0.000,B 0.000,C 90.000,E1 282.007} C_DIS
LIN {X 0.142,Y -441.776,Z 637.561,A 0.000,B 0.000,C 90.000,E1 280.894} C_DIS
LIN {X 0.199,Y -462.097,Z 637.546,A 0.000,B 0.000,C 90.000,E1 278.276} C_DIS
LIN {X 0.014,Y -467.965,Z 637.542,A 0.000,B 0.000,C 90.000,E1 277.530} C_DIS
LIN {X -0.065,Y -473.133,Z 637.538,A 0.000,B 0.000,C 90.000,E1 276.777} C_DIS
LIN {X -0.150,Y -477.490,Z 637.533,A 0.000,B 0.000,C 90.000,E1 276.030} C_DIS
LIN {X -0.008,Y -479.913,Z 637.531,A 0.000,B 0.000,C 90.000,E1 275.511} C_DIS
LIN {X 0.008,Y -482.748,Z 637.526,A 0.000,B 0.000,C 90.000,E1 274.759} C_DIS
LIN {X 0.137,Y -484.171,Z 637.524,A 0.000,B 0.000,C 90.000,E1 274.245} C_DIS
LIN {X -0.171,Y -485.213,Z 637.521,A 0.000,B 0.000,C 90.000,E1 273.784} C_DIS
LIN {X -0.016,Y -485.897,Z 637.518,A 0.000,B 0.000,C 90.000,E1 273.269} C_DIS
LIN {X 0.171,Y -486.288,Z 637.515,A 0.000,B 0.000,C 90.000,E1 272.751} C_DIS
LIN {X -0.148,Y -486.443,Z 637.513,A 0.000,B 0.000,C 90.000,E1 272.293} C_DIS
LIN {X 0.040,Y -486.242,Z 637.510,A 0.000,B 0.000,C 90.000,E1 271.776} C_DIS
LIN {X 0.210,Y -485.740,Z 637.507,A 0.000,B 0.000,C 90.000,E1 271.260} C_DIS
LIN {X -0.103,Y -484.819,Z 637.504,A 0.000,B 0.000,C 90.000,E1 270.802} C_DIS
LIN {X 0.066,Y -483.413,Z 637.502,A 0.000,B 0.000,C 90.000,E1 270.286} C_DIS
LIN {X 0.230,Y -481.436,Z 637.499,A 0.000,B 0.000,C 90.000,E1 269.771} C_DIS
LIN {X -0.096,Y -478.839,Z 637.496,A 0.000,B 0.000,C 90.000,E1 269.312} C_DIS
LIN {X 0.040,Y -475.372,Z 637.493,A 0.000,B 0.000,C 90.000,E1 268.797} C_DIS
LIN {X 0.154,Y -470.989,Z 637.491,A 0.000,B 0.000,C 90.000,E1 268.282} C_DIS
LIN {X -0.205,Y -465.368,Z 637.488,A 0.000,B 0.000,C 90.000,E1 267.822} C_DIS
LIN {X -0.165,Y -462.391,Z 637.487,A 0.000,B 0.000,C 90.000,E1 267.593} C_DIS
LIN {X -0.126,Y -459.011,Z 637.485,A 0.000,B 0.000,C 90.000,E1 267.364} C_DIS
LIN {X 0.208,Y -455.779,Z 637.484,A 0.000,B 0.000,C 90.000,E1 267.135} C_DIS
LIN {X -0.152,Y -448.592,Z 637.482,A 0.000,B 0.000,C 90.000,E1 266.846} C_DIS
LIN {X 0.043,Y -441.072,Z 637.481,A 0.000,B 0.000,C 90.000,E1 266.560} C_DIS
LIN {X -0.167,Y -433.295,Z 637.480,A 0.000,B 0.000,C 90.000,E1 266.388} C_DIS
LIN {X 0.036,Y -424.382,Z 637.479,A 0.000,B 0.000,C 90.000,E1 266.216} C_DIS
LIN {X -0.031,Y -414.963,Z 637.479,A 0.000,B 0.000,C 90.000,E1 266.159} C_DIS
LIN {X -0.038,Y -180.927,Z 637.479,A 0.000,B 0.000,C 90.000,E1 266.159} C_DIS
LIN {X 0.055,Y -180.901,Z 637.474,A 0.000,B 0.000,C 90.000,E1 265.241} C_DIS
LIN {X 0.005,Y -180.226,Z 637.464,A 0.000,B 0.000,C 90.000,E1 263.571} C_DIS
LIN {X -0.042,Y -179.039,Z 637.445,A 0.000,B 0.000,C 90.000,E1 260.208} C_DIS
LIN {X 0.021,Y -178.706,Z 637.441,A 0.000,B 0.000,C 90.000,E1 259.342} C_DIS
LIN {X -0.038,Y -175.755,Z 637.413,A 0.000,B 0.000,C 90.000,E1 254.267} C_DIS
LIN {X -0.035,Y -171.939,Z 637.384,A 0.000,B 0.000,C 90.000,E1 249.135} C_DIS
LIN {X -0.060,Y -171.321,Z 637.379,A 0.000,B 0.000,C 90.000,E1 248.284} C_DIS
LIN {X -0.007,Y -167.578,Z 637.355,A 0.000,B 0.000,C 90.000,E1 243.948} C_DIS
LIN {X -0.067,Y -166.212,Z 637.346,A 0.000,B 0.000,C 90.000,E1 242.231} C_DIS
LIN {X -0.078,Y -162.976,Z 637.326,A 0.000,B 0.000,C 90.000,E1 238.742} C_DIS
LIN {X -0.031,Y -160.889,Z 637.312,A 0.000,B 0.000,C 90.000,E1 236.087} C_DIS
LIN {X -0.052,Y -157.659,Z 637.292,A 0.000,B 0.000,C 90.000,E1 232.557} C_DIS
LIN {X 0.006,Y -155.696,Z 637.277,A 0.000,B 0.000,C 90.000,E1 229.865} C_DIS
LIN {X -0.059,Y -151.960,Z 637.252,A 0.000,B 0.000,C 90.000,E1 225.405} C_DIS
LIN {X -0.042,Y -150.201,Z 637.237,A 0.000,B 0.000,C 90.000,E1 222.690} C_DIS
LIN {X 0.089,Y -146.970,Z 637.212,A 0.000,B 0.000,C 90.000,E1 218.096} C_DIS
LIN {X -0.007,Y -145.557,Z 637.197,A 0.000,B 0.000,C 90.000,E1 215.391} C_DIS
LIN {X -0.008,Y -142.949,Z 637.171,A 0.000,B 0.000,C 90.000,E1 210.797} C_DIS
LIN {X -0.077,Y -141.574,Z 637.151,A 0.000,B 0.000,C 90.000,E1 207.129} C_DIS
LIN {X -0.030,Y -139.414,Z 637.114,A 0.000,B 0.000,C 90.000,E1 200.610} C_DIS
LIN {X 0.023,Y -139.138,Z 637.104,A 0.000,B 0.000,C 90.000,E1 198.725} C_DIS
LIN {X 0.050,Y -138.349,Z 637.057,A 0.000,B 0.000,C 90.000,E1 190.310} C_DIS
LIN {X 0.038,Y -139.494,Z 637.005,A 0.000,B 0.000,C 90.000,E1 180.974} C_DIS
LIN {X -0.022,Y -141.107,Z 636.974,A 0.000,B 0.000,C 90.000,E1 175.412} C_DIS
LIN {X -0.068,Y -142.486,Z 636.959,A 0.000,B 0.000,C 90.000,E1 172.648} C_DIS
LIN {X 0.020,Y -144.737,Z 636.933,A 0.000,B 0.000,C 90.000,E1 167.993} C_DIS
LIN {X -0.030,Y -147.343,Z 636.913,A 0.000,B 0.000,C 90.000,E1 164.338} C_DIS
LIN {X 0.035,Y -150.667,Z 636.888,A 0.000,B 0.000,C 90.000,E1 159.752} C_DIS
LIN {X -0.084,Y -154.146,Z 636.867,A 0.000,B 0.000,C 90.000,E1 156.177} C_DIS
LIN {X 0.051,Y -157.576,Z 636.848,A 0.000,B 0.000,C 90.000,E1 152.538} C_DIS
LIN {X 0.002,Y -161.822,Z 636.828,A 0.000,B 0.000,C 90.000,E1 148.997} C_DIS
LIN {X 0.021,Y -166.013,Z 636.808,A 0.000,B 0.000,C 90.000,E1 145.468} C_DIS
LIN {X 0.013,Y -171.013,Z 636.789,A 0.000,B 0.000,C 90.000,E1 141.984} C_DIS
LIN {X 0.045,Y -175.883,Z 636.770,A 0.000,B 0.000,C 90.000,E1 138.528} C_DIS
LIN {X -0.079,Y -181.487,Z 636.751,A 0.000,B 0.000,C 90.000,E1 135.162} C_DIS
LIN {X 0.057,Y -187.003,Z 636.732,A 0.000,B 0.000,C 90.000,E1 131.757} C_DIS
LIN {X 0.103,Y -191.065,Z 636.720,A 0.000,B 0.000,C 90.000,E1 129.564} C_DIS
LIN {X 0.103,Y -288.584,Z 636.720,A 0.000,B 0.000,C 90.000,E1 129.564} C_DIS
LIN {X -0.054,Y -290.369,Z 636.720,A 0.000,B 0.000,C 90.000,E1 129.564} C_DIS
LIN {X 0.018,Y -295.524,Z 636.718,A 0.000,B 0.000,C 90.000,E1 129.277} C_DIS
LIN {X 0.001,Y -298.722,Z 636.716,A 0.000,B 0.000,C 90.000,E1 128.955} C_DIS
LIN {X -0.019,Y -302.330,Z 636.713,A 0.000,B 0.000,C 90.000,E1 128.382} C_DIS
LIN {X 0.167,Y -303.781,Z 636.711,A 0.000,B 0.000,C 90.000,E1 128.016} C_DIS
LIN {X -0.073,Y -304.923,Z 636.710,A 0.000,B 0.000,C 90.000,E1 127.729} C_DIS
LIN {X 0.030,Y -315.486,Z 636.690,A 0.000,B 0.000,C 90.000,E1 124.119} C_DIS
LIN {X -0.100,Y -325.462,Z 636.674,A 0.000,B 0.000,C 90.000,E1 121.258} C_DIS
LIN {X -0.001,Y -336.758,Z 636.658,A 0.000,B 0.000,C 90.000,E1 118.409} C_DIS
LIN {X -0.064,Y -349.482,Z 636.642,A 0.000,B 0.000,C 90.000,E1 115.643} C_DIS
LIN {X 0.056,Y -362.078,Z 636.629,A 0.000,B 0.000,C 90.000,E1 113.206} C_DIS
LIN {X 0.023,Y -375.980,Z 636.616,A 0.000,B 0.000,C 90.000,E1 110.844} C_DIS
LIN {X -0.068,Y -391.288,Z 636.603,A 0.000,B 0.000,C 90.000,E1 108.544} C_DIS
LIN {X 0.110,Y -408.113,Z 636.590,A 0.000,B 0.000,C 90.000,E1 106.260} C_DIS
LIN {X 0.088,Y -426.579,Z 636.578,A 0.000,B 0.000,C 90.000,E1 104.064} C_DIS
LIN {X 0.173,Y -446.460,Z 636.567,A 0.000,B 0.000,C 90.000,E1 101.951} C_DIS
LIN {X 0.196,Y -466.944,Z 636.556,A 0.000,B 0.000,C 90.000,E1 100.018} C_DIS
LIN {X -0.234,Y -471.948,Z 636.553,A 0.000,B 0.000,C 90.000,E1 99.613} C_DIS
LIN {X 0.205,Y -473.855,Z 636.552,A 0.000,B 0.000,C 90.000,E1 99.321} C_DIS
LIN {X 0.102,Y -475.306,Z 636.551,A 0.000,B 0.000,C 90.000,E1 99.095} C_DIS
LIN {X -0.173,Y -477.299,Z 636.548,A 0.000,B 0.000,C 90.000,E1 98.624} C_DIS
LIN {X -0.041,Y -478.164,Z 636.545,A 0.000,B 0.000,C 90.000,E1 98.106} C_DIS
LIN {X 0.105,Y -478.051,Z 636.542,A 0.000,B 0.000,C 90.000,E1 97.587} C_DIS
LIN {X -0.217,Y -476.945,Z 636.539,A 0.000,B 0.000,C 90.000,E1 97.125} C_DIS
LIN {X 0.123,Y -475.969,Z 636.538,A 0.000,B 0.000,C 90.000,E1 96.834} C_DIS
LIN {X -0.066,Y -474.650,Z 636.537,A 0.000,B 0.000,C 90.000,E1 96.606} C_DIS
LIN {X 0.183,Y -455.677,Z 636.521,A 0.000,B 0.000,C 90.000,E1 93.784} C_DIS
LIN {X 0.100,Y -443.522,Z 636.510,A 0.000,B 0.000,C 90.000,E1 91.718} C_DIS
LIN {X 0.008,Y -433.513,Z 636.499,A 0.000,B 0.000,C 90.000,E1 89.885} C_DIS
LIN {X -0.121,Y -426.059,Z 636.492,A 0.000,B 0.000,C 90.000,E1 88.568} C_DIS
LIN {X -0.111,Y -415.151,Z 636.481,A 0.000,B 0.000,C 90.000,E1 86.674} C_DIS
LIN {X 0.082,Y -404.221,Z 636.471,A 0.000,B 0.000,C 90.000,E1 84.723} C_DIS
LIN {X -0.144,Y -389.130,Z 636.455,A 0.000,B 0.000,C 90.000,E1 81.951} C_DIS
LIN {X 0.058,Y -376.209,Z 636.441,A 0.000,B 0.000,C 90.000,E1 79.342} C_DIS
LIN {X 0.133,Y -365.055,Z 636.428,A 0.000,B 0.000,C 90.000,E1 76.992} C_DIS
LIN {X -0.023,Y -349.190,Z 636.408,A 0.000,B 0.000,C 90.000,E1 73.433} C_DIS
LIN {X 0.010,Y -338.096,Z 636.393,A 0.000,B 0.000,C 90.000,E1 70.678} C_DIS
LIN {X 0.113,Y -325.463,Z 636.374,A 0.000,B 0.000,C 90.000,E1 67.230} C_DIS
LIN {X -0.016,Y -313.093,Z 636.352,A 0.000,B 0.000,C 90.000,E1 63.435} C_DIS
LIN {X -0.088,Y -303.714,Z 636.334,A 0.000,B 0.000,C 90.000,E1 60.205} C_DIS
LIN {X -0.114,Y -295.013,Z 636.316,A 0.000,B 0.000,C 90.000,E1 56.914} C_DIS
LIN {X 0.104,Y -288.422,Z 636.301,A 0.000,B 0.000,C 90.000,E1 54.196} C_DIS
LIN {X -0.137,Y -282.057,Z 636.286,A 0.000,B 0.000,C 90.000,E1 51.537} C_DIS
LIN {X -0.016,Y -277.020,Z 636.275,A 0.000,B 0.000,C 90.000,E1 49.461} C_DIS
LIN {X -0.009,Y -273.402,Z 636.267,A 0.000,B 0.000,C 90.000,E1 48.081} C_DIS
LIN {X -0.047,Y -269.579,Z 636.259,A 0.000,B 0.000,C 90.000,E1 46.701} C_DIS
LIN {X -0.142,Y -265.470,Z 636.252,A 0.000,B 0.000,C 90.000,E1 45.324} C_DIS
LIN {X 0.002,Y -258.922,Z 636.240,A 0.000,B 0.000,C 90.000,E1 43.176} C_DIS
LIN {X 0.034,Y -249.919,Z 636.224,A 0.000,B 0.000,C 90.000,E1 40.297} C_DIS
LIN {X -0.057,Y -239.392,Z 636.204,A 0.000,B 0.000,C 90.000,E1 36.664} C_DIS
LIN {X 0.055,Y -231.718,Z 636.187,A 0.000,B 0.000,C 90.000,E1 33.658} C_DIS
LIN {X -0.085,Y -224.816,Z 636.170,A 0.000,B 0.000,C 90.000,E1 30.669} C_DIS
LIN {X -0.041,Y -218.556,Z 636.153,A 0.000,B 0.000,C 90.000,E1 27.590} C_DIS
LIN {X 0.033,Y -213.123,Z 636.136,A 0.000,B 0.000,C 90.000,E1 24.463} C_DIS
LIN {X -0.066,Y -207.396,Z 636.114,A 0.000,B 0.000,C 90.000,E1 20.556} C_DIS
LIN {X 0.020,Y -202.875,Z 636.092,A 0.000,B 0.000,C 90.000,E1 16.551} C_DIS
LIN {X 0.011,Y -199.384,Z 636.070,A 0.000,B 0.000,C 90.000,E1 12.535} C_DIS
LIN {X -0.088,Y -196.235,Z 636.038,A 0.000,B 0.000,C 90.000,E1 6.891} C_DIS
LIN {X 0.020,Y -197.227,Z 635.957,A 0.000,B 0.000,C 90.000,E1 352.186} C_DIS
LIN {X -0.100,Y -200.416,Z 635.930,A 0.000,B 0.000,C 90.000,E1 347.353} C_DIS
LIN {X -0.091,Y -204.223,Z 635.907,A 0.000,B 0.000,C 90.000,E1 343.323} C_DIS
LIN {X -0.043,Y -208.912,Z 635.885,A 0.000,B 0.000,C 90.000,E1 339.316} C_DIS
LIN {X -0.010,Y -214.449,Z 635.863,A 0.000,B 0.000,C 90.000,E1 335.357} C_DIS
LIN {X 0.063,Y -220.671,Z 635.841,A 0.000,B 0.000,C 90.000,E1 331.435} C_DIS
LIN {X 0.076,Y -227.540,Z 635.820,A 0.000,B 0.000,C 90.000,E1 327.582} C_DIS
LIN {X 0.091,Y -234.921,Z 635.799,A 0.000,B 0.000,C 90.000,E1 323.783} C_DIS
LIN {X -0.007,Y -242.902,Z 635.778,A 0.000,B 0.000,C 90.000,E1 320.070} C_DIS
LIN {X 0.065,Y -251.727,Z 635.758,A 0.000,B 0.000,C 90.000,E1 316.377} C_DIS
LIN {X 0.053,Y -261.599,Z 635.738,A 0.000,B 0.000,C 90.000,E1 312.771} C_DIS
LIN {X 0.174,Y -271.675,Z 635.720,A 0.000,B 0.000,C 90.000,E1 309.564} C_DIS
LIN {X -0.118,Y -282.951,Z 635.703,A 0.000,B 0.000,C 90.000,E1 306.503} C_DIS
LIN {X 0.027,Y -297.008,Z 635.684,A 0.000,B 0.000,C 90.000,E1 303.086} C_DIS
LIN {X -0.054,Y -311.045,Z 635.667,A 0.000,B 0.000,C 90.000,E1 300.129} C_DIS
LIN {X 0.060,Y -322.764,Z 635.655,A 0.000,B 0.000,C 90.000,E1 297.847} C_DIS
LIN {X 0.000,Y -334.784,Z 635.642,A 0.000,B 0.000,C 90.000,E1 295.643} C_DIS
LIN {X 0.085,Y -349.261,Z 635.629,A 0.000,B 0.000,C 90.000,E1 293.153} C_DIS
LIN {X -0.107,Y -368.696,Z 635.612,A 0.000,B 0.000,C 90.000,E1 290.174} C_DIS
LIN {X -0.135,Y -383.717,Z 635.601,A 0.000,B 0.000,C 90.000,E1 288.127} C_DIS
LIN {X -0.138,Y -402.216,Z 635.588,A 0.000,B 0.000,C 90.000,E1 285.843} C_DIS
LIN {X 0.031,Y -413.764,Z 635.580,A 0.000,B 0.000,C 90.000,E1 284.426} C_DIS
LIN {X -0.032,Y -424.875,Z 635.573,A 0.000,B 0.000,C 90.000,E1 283.063} C_DIS
LIN {X -0.022,Y -435.564,Z 635.565,A 0.000,B 0.000,C 90.000,E1 281.715} C_DIS
LIN {X 0.138,Y -445.753,Z 635.558,A 0.000,B 0.000,C 90.000,E1 280.366} C_DIS
LIN {X 0.197,Y -461.950,Z 635.546,A 0.000,B 0.000,C 90.000,E1 278.276} C_DIS
LIN {X 0.010,Y -467.808,Z 635.542,A 0.000,B 0.000,C 90.000,E1 277.530} C_DIS
LIN {X -0.070,Y -473.004,Z 635.538,A 0.000,B 0.000,C 90.000,E1 276.777} C_DIS
LIN {X -0.105,Y -477.372,Z 635.533,A 0.000,B 0.000,C 90.000,E1 276.024} C_DIS
LIN {X -0.158,Y -480.819,Z 635.529,A 0.000,B 0.000,C 90.000,E1 275.277} C_DIS
LIN {X 0.000,Y -482.601,Z 635.526,A 0.000,B 0.000,C 90.000,E1 274.759} C_DIS
LIN {X 0.128,Y -484.043,Z 635.524,A 0.000,B 0.000,C 90.000,E1 274.245} C_DIS
LIN {X -0.180,Y -485.109,Z 635.521,A 0.000,B 0.000,C 90.000,E1 273.784} C_DIS
LIN {X -0.027,Y -485.801,Z 635.518,A 0.000,B 0.000,C 90.000,E1 273.269} C_DIS
LIN {X 0.159,Y -486.217,Z 635.515,A 0.000,B 0.000,C 90.000,E1 272.751} C_DIS
LIN {X -0.159,Y -486.350,Z 635.513,A 0.000,B 0.000,C 90.000,E1 272.293} C_DIS
LIN {X 0.028,Y -486.172,Z 635.510,A 0.000,B 0.000,C 90.000,E1 271.776} C_DIS
LIN {X 0.198,Y -485.693,Z 635.507,A 0.000,B 0.000,C 90.000,E1 271.260} C_DIS
LIN {X -0.116,Y -484.800,Z 635.504,A 0.000,B 0.000,C 90.000,E1 270.802} C_DIS
LIN {X 0.053,Y -483.405,Z 635.502,A 0.000,B 0.000,C 90.000,E1 270.286} C_DIS
LIN {X 0.217,Y -481.414,Z 635.499,A 0.000,B 0.000,C 90.000,E1 269.771} C_DIS
LIN {X 0.054,Y -480.221,Z 635.497,A 0.000,B 0.000,C 90.000,E1 269.542} C_DIS
LIN {X 0.198,Y -477.221,Z 635.495,A 0.000,B 0.000,C 90.000,E1 269.026} C_DIS
LIN {X -0.152,Y -473.316,Z 635.492,A 0.000,B 0.000,C 90.000,E1 268.568} C_DIS
LIN {X 0.141,Y -471.003,Z 635.491,A 0.000,B 0.000,C 90.000,E1 268.282} C_DIS
LIN {X -0.032,Y -468.355,Z 635.489,A 0.000,B 0.000,C 90.000,E1 268.051} C_DIS
LIN {X -0.218,Y -465.393,Z 635.488,A 0.000,B 0.000,C 90.000,E1 267.822} C_DIS
LIN {X -0.129,Y -459.024,Z 635.485,A 0.000,B 0.000,C 90.000,E1 267.364} C_DIS
LIN {X 0.202,Y -455.778,Z 635.484,A 0.000,B 0.000,C 90.000,E1 267.135} C_DIS
LIN {X 0.077,Y -452.052,Z 635.483,A 0.000,B 0.000,C 90.000,E1 266.963} C_DIS
LIN {X 0.001,Y -444.517,Z 635.482,A 0.000,B 0.000,C 90.000,E1 266.674} C_DIS
LIN {X 0.021,Y -436.838,Z 635.480,A 0.000,B 0.000,C 90.000,E1 266.445} C_DIS
LIN {X 0.017,Y -428.389,Z 635.479,A 0.000,B 0.000,C 90.000,E1 266.274} C_DIS
LIN {X -0.202,Y -421.262,Z 635.479,A 0.000,B 0.000,C 90.000,E1 266.216} C_DIS
LIN {X -0.108,Y -411.759,Z 635.479,A 0.000,B 0.000,C 90.000,E1 266.159} C_DIS
LIN {X -0.072,Y -180.926,Z 635.479,A 0.000,B 0.000,C 90.000,E1 266.159} C_DIS
LIN {X 0.042,Y -180.901,Z 635.474,A 0.000,B 0.000,C 90.000,E1 265.241} C_DIS
LIN {X -0.009,Y -180.223,Z 635.464,A 0.000,B 0.000,C 90.000,E1 263.571} C_DIS
LIN {X -0.055,Y -179.039,Z 635.445,A 0.000,B 0.000,C 90.000,E1 260.208} C_DIS
LIN {X 0.008,Y -178.704,Z 635.441,A 0.000,B 0.000,C 90.000,E1 259.342} C_DIS
LIN {X -0.052,Y -175.752,Z 635.412,A 0.000,B 0.000,C 90.000,E1 254.267} C_DIS
LIN {X -0.048,Y -171.936,Z 635.384,A 0.000,B 0.000,C 90.000,E1 249.135} C_DIS
LIN {X -0.072,Y -171.316,Z 635.379,A 0.000,B 0.000,C 90.000,E1 248.284} C_DIS
LIN {X -0.019,Y -167.575,Z 635.355,A 0.000,B 0.000,C 90.000,E1 243.948} C_DIS
LIN {X -0.080,Y -166.207,Z 635.346,A 0.000,B 0.000,C 90.000,E1 242.231} C_DIS
LIN {X -0.091,Y -162.972,Z 635.326,A 0.000,B 0.000,C 90.000,E1 238.742} C_DIS
LIN {X -0.044,Y -160.884,Z 635.312,A 0.000,B 0.000,C 90.000,E1 236.087} C_DIS
LIN {X -0.065,Y -157.655,Z 635.292,A 0.000,B 0.000,C 90.000,E1 232.557} C_DIS
LIN {X 0.094,Y -155.692,Z 635.277,A 0.000,B 0.000,C 90.000,E1 229.828} C_DIS
LIN {X -0.071,Y -151.956,Z 635.252,A 0.000,B 0.000,C 90.000,E1 225.405} C_DIS
LIN {X -0.053,Y -150.197,Z 635.237,A 0.000,B 0.000,C 90.000,E1 222.690} C_DIS
LIN {X 0.077,Y -146.967,Z 635.212,A 0.000,B 0.000,C 90.000,E1 218.096} C_DIS
LIN {X -0.020,Y -145.554,Z 635.197,A 0.000,B 0.000,C 90.000,E1 215.391} C_DIS
LIN {X -0.020,Y -142.947,Z 635.171,A 0.000,B 0.000,C 90.000,E1 210.797} C_DIS
LIN {X 0.037,Y -141.573,Z 635.151,A 0.000,B 0.000,C 90.000,E1 207.078} C_DIS
LIN {X -0.041,Y -139.413,Z 635.114,A 0.000,B 0.000,C 90.000,E1 200.610} C_DIS
LIN {X 0.012,Y -139.136,Z 635.104,A 0.000,B 0.000,C 90.000,E1 198.725} C_DIS
LIN {X 0.038,Y -138.349,Z 635.057,A 0.000,B 0.000,C 90.000,E1 190.310} C_DIS
LIN {X 0.026,Y -139.495,Z 635.005,A 0.000,B 0.000,C 90.000,E1 180.974} C_DIS
LIN {X -0.034,Y -141.110,Z 634.974,A 0.000,B 0.000,C 90.000,E1 175.412} C_DIS
LIN {X 0.061,Y -142.489,Z 634.959,A 0.000,B 0.000,C 90.000,E1 172.591} C_DIS
LIN {X 0.008,Y -144.740,Z 634.933,A 0.000,B 0.000,C 90.000,E1 167.993} C_DIS
LIN {X -0.041,Y -147.347,Z 634.913,A 0.000,B 0.000,C 90.000,E1 164.338} C_DIS
LIN {X 0.023,Y -150.671,Z 634.888,A 0.000,B 0.000,C 90.000,E1 159.752} C_DIS
LIN {X -0.096,Y -154.151,Z 634.867,A 0.000,B 0.000,C 90.000,E1 156.177} C_DIS
LIN {X 0.038,Y -157.581,Z 634.848,A 0.000,B 0.000,C 90.000,E1 152.538} C_DIS
LIN {X -0.010,Y -161.828,Z 634.828,A 0.000,B 0.000,C 90.000,E1 148.997} C_DIS
LIN {X 0.008,Y -166.019,Z 634.808,A 0.000,B 0.000,C 90.000,E1 145.468} C_DIS
LIN {X 0.000,Y -171.019,Z 634.789,A 0.000,B 0.000,C 90.000,E1 141.984} C_DIS
LIN {X 0.031,Y -175.890,Z 634.770,A 0.000,B 0.000,C 90.000,E1 138.528} C_DIS
LIN {X -0.093,Y -181.494,Z 634.751,A 0.000,B 0.000,C 90.000,E1 135.162} C_DIS
LIN {X 0.043,Y -187.011,Z 634.732,A 0.000,B 0.000,C 90.000,E1 131.757} C_DIS
LIN {X 0.089,Y -191.072,Z 634.720,A 0.000,B 0.000,C 90.000,E1 129.564} C_DIS
LIN {X 0.082,Y -288.578,Z 634.720,A 0.000,B 0.000,C 90.000,E1 129.564} C_DIS
LIN {X -0.076,Y -290.362,Z 634.720,A 0.000,B 0.000,C 90.000,E1 129.564} C_DIS
LIN {X -0.002,Y -295.515,Z 634.718,A 0.000,B 0.000,C 90.000,E1 129.277} C_DIS
LIN {X -0.022,Y -298.713,Z 634.716,A 0.000,B 0.000,C 90.000,E1 128.955} C_DIS
LIN {X -0.041,Y -302.321,Z 634.713,A 0.000,B 0.000,C 90.000,E1 128.382} C_DIS
LIN {X 0.146,Y -303.772,Z 634.711,A 0.000,B 0.000,C 90.000,E1 128.016} C_DIS
LIN {X -0.095,Y -304.914,Z 634.710,A 0.000,B 0.000,C 90.000,E1 127.729} C_DIS
LIN {X 0.006,Y -315.479,Z 634.690,A 0.000,B 0.000,C 90.000,E1 124.119} C_DIS
LIN {X -0.123,Y -325.456,Z 634.674,A 0.000,B 0.000,C 90.000,E1 121.258} C_DIS
LIN {X -0.026,Y -336.754,Z 634.658,A 0.000,B 0.000,C 90.000,E1 118.409} C_DIS
LIN {X -0.090,Y -349.480,Z 634.642,A 0.000,B 0.000,C 90.000,E1 115.643} C_DIS
LIN {X 0.029,Y -362.078,Z 634.629,A 0.000,B 0.000,C 90.000,E1 113.206} C_DIS
LIN {X -0.006,Y -375.982,Z 634.616,A 0.000,B 0.000,C 90.000,E1 110.844} C_DIS
LIN {X -0.097,Y -391.293,Z 634.603,A 0.000,B 0.000,C 90.000,E1 108.544} C_DIS
LIN {X 0.079,Y -408.121,Z 634.590,A 0.000,B 0.000,C 90.000,E1 106.260} C_DIS
LIN {X 0.056,Y -426.590,Z 634.578,A 0.000,B 0.000,C 90.000,E1 104.064} C_DIS
LIN {X 0.142,Y -446.472,Z 634.566,A 0.000,B 0.000,C 90.000,E1 101.951} C_DIS
LIN {X 0.164,Y -466.957,Z 634.556,A 0.000,B 0.000,C 90.000,E1 100.018} C_DIS
LIN {X 0.201,Y -471.979,Z 634.553,A 0.000,B 0.000,C 90.000,E1 99.557} C_DIS
LIN {X 0.183,Y -473.896,Z 634.552,A 0.000,B 0.000,C 90.000,E1 99.321} C_DIS
LIN {X 0.089,Y -475.356,Z 634.551,A 0.000,B 0.000,C 90.000,E1 99.095} C_DIS
LIN {X -0.186,Y -477.376,Z 634.548,A 0.000,B 0.000,C 90.000,E1 98.624} C_DIS
LIN {X -0.054,Y -478.261,Z 634.545,A 0.000,B 0.000,C 90.000,E1 98.106} C_DIS
LIN {X 0.091,Y -478.166,Z 634.542,A 0.000,B 0.000,C 90.000,E1 97.587} C_DIS
LIN {X -0.230,Y -477.080,Z 634.539,A 0.000,B 0.000,C 90.000,E1 97.125} C_DIS
LIN {X 0.111,Y -476.116,Z 634.538,A 0.000,B 0.000,C 90.000,E1 96.834} C_DIS
LIN {X -0.078,Y -474.811,Z 634.537,A 0.000,B 0.000,C 90.000,E1 96.606} C_DIS
LIN {X 0.177,Y -455.776,Z 634.521,A 0.000,B 0.000,C 90.000,E1 93.784} C_DIS
LIN {X 0.096,Y -443.631,Z 634.510,A 0.000,B 0.000,C 90.000,E1 91.718} C_DIS
LIN {X 0.005,Y -433.620,Z 634.499,A 0.000,B 0.000,C 90.000,E1 89.885} C_DIS
LIN {X -0.122,Y -426.152,Z 634.492,A 0.000,B 0.000,C 90.000,E1 88.568} C_DIS
LIN {X -0.109,Y -415.260,Z 634.481,A 0.000,B 0.000,C 90.000,E1 86.674} C_DIS
LIN {X 0.179,Y -402.775,Z 634.469,A 0.000,B 0.000,C 90.000,E1 84.432} C_DIS
LIN {X -0.082,Y -387.785,Z 634.454,A 0.000,B 0.000,C 90.000,E1 81.659} C_DIS
LIN {X 0.079,Y -374.902,Z 634.439,A 0.000,B 0.000,C 90.000,E1 79.050} C_DIS
LIN {X 0.122,Y -363.769,Z 634.426,A 0.000,B 0.000,C 90.000,E1 76.700} C_DIS
LIN {X -0.009,Y -349.302,Z 634.408,A 0.000,B 0.000,C 90.000,E1 73.433} C_DIS
LIN {X 0.139,Y -339.431,Z 634.394,A 0.000,B 0.000,C 90.000,E1 70.967} C_DIS
LIN {X 0.134,Y -325.598,Z 634.374,A 0.000,B 0.000,C 90.000,E1 67.230} C_DIS
LIN {X 0.009,Y -313.267,Z 634.352,A 0.000,B 0.000,C 90.000,E1 63.435} C_DIS
LIN {X -0.057,Y -303.891,Z 634.334,A 0.000,B 0.000,C 90.000,E1 60.205} C_DIS
LIN {X -0.079,Y -295.183,Z 634.316,A 0.000,B 0.000,C 90.000,E1 56.914} C_DIS
LIN {X 0.142,Y -288.581,Z 634.301,A 0.000,B 0.000,C 90.000,E1 54.196} C_DIS
LIN {X 0.034,Y -283.836,Z 634.290,A 0.000,B 0.000,C 90.000,E1 52.190} C_DIS
LIN {X 0.009,Y -278.890,Z 634.279,A 0.000,B 0.000,C 90.000,E1 50.150} C_DIS
LIN {X 0.035,Y -273.586,Z 634.267,A 0.000,B 0.000,C 90.000,E1 48.081} C_DIS
LIN {X -0.001,Y -269.746,Z 634.259,A 0.000,B 0.000,C 90.000,E1 46.701} C_DIS
LIN {X -0.095,Y -265.633,Z 634.252,A 0.000,B 0.000,C 90.000,E1 45.324} C_DIS
LIN {X 0.050,Y -259.084,Z 634.240,A 0.000,B 0.000,C 90.000,E1 43.176} C_DIS
LIN {X -0.070,Y -250.049,Z 634.224,A 0.000,B 0.000,C 90.000,E1 40.334} C_DIS
LIN {X 0.002,Y -239.522,Z 634.204,A 0.000,B 0.000,C 90.000,E1 36.664} C_DIS
LIN {X -0.078,Y -231.848,Z 634.187,A 0.000,B 0.000,C 90.000,E1 33.706} C_DIS
LIN {X -0.023,Y -224.962,Z 634.170,A 0.000,B 0.000,C 90.000,E1 30.669} C_DIS
LIN {X 0.022,Y -218.680,Z 634.153,A 0.000,B 0.000,C 90.000,E1 27.590} C_DIS
LIN {X -0.096,Y -213.237,Z 634.136,A 0.000,B 0.000,C 90.000,E1 24.515} C_DIS
LIN {X 0.000,Y -207.500,Z 634.114,A 0.000,B 0.000,C 90.000,E1 20.556} C_DIS
LIN {X 0.031,Y -202.970,Z 634.092,A 0.000,B 0.000,C 90.000,E1 16.567} C_DIS
LIN {X 0.081,Y -199.466,Z 634.070,A 0.000,B 0.000,C 90.000,E1 12.535} C_DIS
LIN {X -0.016,Y -196.298,Z 634.038,A 0.000,B 0.000,C 90.000,E1 6.891} C_DIS
LIN {X 0.024,Y -197.284,Z 633.957,A 0.000,B 0.000,C 90.000,E1 352.186} C_DIS
LIN {X -0.094,Y -200.482,Z 633.930,A 0.000,B 0.000,C 90.000,E1 347.353} C_DIS
LIN {X -0.083,Y -204.290,Z 633.907,A 0.000,B 0.000,C 90.000,E1 343.323} C_DIS
LIN {X -0.033,Y -208.967,Z 633.885,A 0.000,B 0.000,C 90.000,E1 339.316} C_DIS
LIN {X 0.003,Y -214.509,Z 633.863,A 0.000,B 0.000,C 90.000,E1 335.357} C_DIS
LIN {X 0.077,Y -220.710,Z 633.841,A 0.000,B 0.000,C 90.000,E1 331.435} C_DIS
LIN {X 0.091,Y -227.548,Z 633.820,A 0.000,B 0.000,C 90.000,E1 327.582} C_DIS
LIN {X -0.082,Y -234.932,Z 633.799,A 0.000,B 0.000,C 90.000,E1 323.829} C_DIS
LIN {X 0.011,Y -242.902,Z 633.778,A 0.000,B 0.000,C 90.000,E1 320.070} C_DIS
LIN {X 0.082,Y -251.714,Z 633.758,A 0.000,B 0.000,C 90.000,E1 316.377} C_DIS
LIN {X 0.072,Y -261.540,Z 633.738,A 0.000,B 0.000,C 90.000,E1 312.771} C_DIS
LIN {X 0.018,Y -271.600,Z 633.720,A 0.000,B 0.000,C 90.000,E1 309.600} C_DIS
LIN {X -0.101,Y -282.867,Z 633.703,A 0.000,B 0.000,C 90.000,E1 306.503} C_DIS
LIN {X 0.041,Y -296.906,Z 633.684,A 0.000,B 0.000,C 90.000,E1 303.086} C_DIS
LIN {X -0.042,Y -310.969,Z 633.667,A 0.000,B 0.000,C 90.000,E1 300.129} C_DIS
LIN {X 0.154,Y -324.360,Z 633.653,A 0.000,B 0.000,C 90.000,E1 297.513} C_DIS
LIN {X -0.024,Y -336.433,Z 633.641,A 0.000,B 0.000,C 90.000,E1 295.335} C_DIS
LIN {X -0.215,Y -351.030,Z 633.627,A 0.000,B 0.000,C 90.000,E1 292.898} C_DIS
LIN {X -0.104,Y -368.648,Z 633.612,A 0.000,B 0.000,C 90.000,E1 290.174} C_DIS
LIN {X -0.134,Y -383.677,Z 633.601,A 0.000,B 0.000,C 90.000,E1 288.127} C_DIS
LIN {X -0.137,Y -402.163,Z 633.588,A 0.000,B 0.000,C 90.000,E1 285.843} C_DIS
LIN {X 0.030,Y -413.701,Z 633.580,A 0.000,B 0.000,C 90.000,E1 284.426} C_DIS
LIN {X -0.033,Y -424.810,Z 633.573,A 0.000,B 0.000,C 90.000,E1 283.063} C_DIS
LIN {X -0.024,Y -435.517,Z 633.565,A 0.000,B 0.000,C 90.000,E1 281.715} C_DIS
LIN {X 0.135,Y -445.723,Z 633.558,A 0.000,B 0.000,C 90.000,E1 280.366} C_DIS
LIN {X 0.193,Y -461.849,Z 633.546,A 0.000,B 0.000,C 90.000,E1 278.276} C_DIS
LIN {X -0.163,Y -469.459,Z 633.540,A 0.000,B 0.000,C 90.000,E1 277.296} C_DIS
LIN {X 0.242,Y -474.398,Z 633.536,A 0.000,B 0.000,C 90.000,E1 276.486} C_DIS
LIN {X -0.112,Y -477.238,Z 633.533,A 0.000,B 0.000,C 90.000,E1 276.024} C_DIS
LIN {X -0.166,Y -480.697,Z 633.529,A 0.000,B 0.000,C 90.000,E1 275.277} C_DIS
LIN {X -0.008,Y -482.511,Z 633.526,A 0.000,B 0.000,C 90.000,E1 274.759} C_DIS
LIN {X 0.118,Y -483.942,Z 633.524,A 0.000,B 0.000,C 90.000,E1 274.245} C_DIS
LIN {X -0.190,Y -485.008,Z 633.521,A 0.000,B 0.000,C 90.000,E1 273.784} C_DIS
LIN {X -0.038,Y -485.735,Z 633.518,A 0.000,B 0.000,C 90.000,E1 273.269} C_DIS
LIN {X 0.148,Y -486.137,Z 633.515,A 0.000,B 0.000,C 90.000,E1 272.751} C_DIS
LIN {X -0.172,Y -486.287,Z 633.513,A 0.000,B 0.000,C 90.000,E1 272.293} C_DIS
LIN {X 0.015,Y -486.155,Z 633.510,A 0.000,B 0.000,C 90.000,E1 271.776} C_DIS
LIN {X 0.186,Y -485.674,Z 633.507,A 0.000,B 0.000,C 90.000,E1 271.260} C_DIS
LIN {X -0.128,Y -484.780,Z 633.504,A 0.000,B 0.000,C 90.000,E1 270.802} C_DIS
LIN {X 0.040,Y -483.392,Z 633.502,A 0.000,B 0.000,C 90.000,E1 270.286} C_DIS
LIN {X 0.204,Y -481.470,Z 633.499,A 0.000,B 0.000,C 90.000,E1 269.771} C_DIS
LIN {X -0.122,Y -478.834,Z 633.496,A 0.000,B 0.000,C 90.000,E1 269.312} C_DIS
LIN {X 0.013,Y -475.409,Z 633.493,A 0.000,B 0.000,C 90.000,E1 268.797} C_DIS
LIN {X 0.128,Y -471.004,Z 633.491,A 0.000,B 0.000,C 90.000,E1 268.282} C_DIS
LIN {X -0.045,Y -468.378,Z 633.489,A 0.000,B 0.000,C 90.000,E1 268.051} C_DIS
LIN {X 0.234,Y -465.437,Z 633.488,A 0.000,B 0.000,C 90.000,E1 267.764} C_DIS
LIN {X -0.196,Y -462.429,Z 633.487,A 0.000,B 0.000,C 90.000,E1 267.593} C_DIS
LIN {X 0.195,Y -455.782,Z 633.484,A 0.000,B 0.000,C 90.000,E1 267.135} C_DIS
LIN {X -0.148,Y -448.668,Z 633.482,A 0.000,B 0.000,C 90.000,E1 266.846} C_DIS
LIN {X 0.037,Y -441.087,Z 633.481,A 0.000,B 0.000,C 90.000,E1 266.560} C_DIS
LIN {X -0.200,Y -433.167,Z 633.480,A 0.000,B 0.000,C 90.000,E1 266.388} C_DIS
LIN {X -0.015,Y -424.120,Z 633.479,A 0.000,B 0.000,C 90.000,E1 266.216} C_DIS
LIN {X -0.027,Y -416.872,Z 633.479,A 0.000,B 0.000,C 90.000,E1 266.159} C_DIS
LIN {X -0.141,Y -412.765,Z 633.479,A 0.000,B 0.000,C 90.000,E1 266.159} C_DIS
LIN {X -0.086,Y -180.926,Z 633.479,A 0.000,B 0.000,C 90.000,E1 266.159} C_DIS
LIN {X 0.026,Y -180.900,Z 633.474,A 0.000,B 0.000,C 90.000,E1 265.241} C_DIS
LIN {X -0.024,Y -180.221,Z 633.464,A 0.000,B 0.000,C 90.000,E1 263.571} C_DIS
LIN {X -0.071,Y -179.037,Z 633.445,A 0.000,B 0.000,C 90.000,E1 260.208} C_DIS
LIN {X -0.008,Y -178.701,Z 633.441,A 0.000,B 0.000,C 90.000,E1 259.342} C_DIS
LIN {X 0.102,Y -175.749,Z 633.412,A 0.000,B 0.000,C 90.000,E1 254.212} C_DIS
LIN {X 0.097,Y -171.933,Z 633.384,A 0.000,B 0.000,C 90.000,E1 249.082} C_DIS
LIN {X -0.088,Y -171.312,Z 633.379,A 0.000,B 0.000,C 90.000,E1 248.284} C_DIS
LIN {X -0.034,Y -167.572,Z 633.355,A 0.000,B 0.000,C 90.000,E1 243.948} C_DIS
LIN {X -0.095,Y -166.201,Z 633.346,A 0.000,B 0.000,C 90.000,E1 242.231} C_DIS
LIN {X -0.021,Y -162.967,Z 633.326,A 0.000,B 0.000,C 90.000,E1 238.712} C_DIS
LIN {X -0.058,Y -160.879,Z 633.311,A 0.000,B 0.000,C 90.000,E1 236.087} C_DIS
LIN {X -0.080,Y -157.651,Z 633.292,A 0.000,B 0.000,C 90.000,E1 232.557} C_DIS
LIN {X 0.078,Y -155.688,Z 633.277,A 0.000,B 0.000,C 90.000,E1 229.828} C_DIS
LIN {X -0.085,Y -151.953,Z 633.252,A 0.000,B 0.000,C 90.000,E1 225.405} C_DIS
LIN {X -0.068,Y -150.193,Z 633.237,A 0.000,B 0.000,C 90.000,E1 222.690} C_DIS
LIN {X 0.063,Y -146.964,Z 633.212,A 0.000,B 0.000,C 90.000,E1 218.096} C_DIS
LIN {X -0.034,Y -145.551,Z 633.197,A 0.000,B 0.000,C 90.000,E1 215.391} C_DIS
LIN {X -0.033,Y -142.945,Z 633.171,A 0.000,B 0.000,C 90.000,E1 210.797} C_DIS
LIN {X 0.023,Y -141.570,Z 633.151,A 0.000,B 0.000,C 90.000,E1 207.078} C_DIS
LIN {X -0.055,Y -139.412,Z 633.114,A 0.000,B 0.000,C 90.000,E1 200.610} C_DIS
LIN {X -0.003,Y -139.134,Z 633.104,A 0.000,B 0.000,C 90.000,E1 198.725} C_DIS
LIN {X 0.025,Y -138.349,Z 633.057,A 0.000,B 0.000,C 90.000,E1 190.310} C_DIS
LIN {X 0.012,Y -139.495,Z 633.005,A 0.000,B 0.000,C 90.000,E1 180.974} C_DIS
LIN {X -0.048,Y -141.112,Z 632.974,A 0.000,B 0.000,C 90.000,E1 175.412} C_DIS
LIN {X 0.047,Y -142.492,Z 632.959,A 0.000,B 0.000,C 90.000,E1 172.591} C_DIS
LIN {X -0.006,Y -144.744,Z 632.933,A 0.000,B 0.000,C 90.000,E1 167.993} C_DIS
LIN {X -0.056,Y -147.351,Z 632.913,A 0.000,B 0.000,C 90.000,E1 164.338} C_DIS
LIN {X 0.009,Y -150.676,Z 632.888,A 0.000,B 0.000,C 90.000,E1 159.752} C_DIS
LIN {X 0.029,Y -154.155,Z 632.867,A 0.000,B 0.000,C 90.000,E1 156.125} C_DIS
LIN {X 0.023,Y -157.587,Z 632.847,A 0.000,B 0.000,C 90.000,E1 152.538} C_DIS
LIN {X -0.026,Y -161.835,Z 632.828,A 0.000,B 0.000,C 90.000,E1 148.997} C_DIS
LIN {X -0.008,Y -166.026,Z 632.808,A 0.000,B 0.000,C 90.000,E1 145.468} C_DIS
LIN {X -0.016,Y -171.027,Z 632.789,A 0.000,B 0.000,C 90.000,E1 141.984} C_DIS
LIN {X 0.015,Y -175.898,Z 632.770,A 0.000,B 0.000,C 90.000,E1 138.528} C_DIS
LIN {X 0.020,Y -181.501,Z 632.751,A 0.000,B 0.000,C 90.000,E1 135.121} C_DIS
LIN {X 0.026,Y -187.019,Z 632.732,A 0.000,B 0.000,C 90.000,E1 131.757} C_DIS
LIN {X 0.072,Y -191.081,Z 632.720,A 0.000,B 0.000,C 90.000,E1 129.564} C_DIS
LIN {X 0.057,Y -288.617,Z 632.720,A 0.000,B 0.000,C 90.000,E1 129.564} C_DIS
LIN {X -0.102,Y -290.370,Z 632.720,A 0.000,B 0.000,C 90.000,E1 129.564} C_DIS
LIN {X -0.028,Y -295.512,Z 632.718,A 0.000,B 0.000,C 90.000,E1 129.277} C_DIS
LIN {X -0.050,Y -298.713,Z 632.716,A 0.000,B 0.000,C 90.000,E1 128.955} C_DIS
LIN {X -0.073,Y -302.320,Z 632.713,A 0.000,B 0.000,C 90.000,E1 128.382} C_DIS
LIN {X 0.113,Y -303.770,Z 632.711,A 0.000,B 0.000,C 90.000,E1 128.016} C_DIS
LIN {X -0.127,Y -304.911,Z 632.709,A 0.000,B 0.000,C 90.000,E1 127.729} C_DIS
LIN {X -0.027,Y -315.478,Z 632.690,A 0.000,B 0.000,C 90.000,E1 124.119} C_DIS
LIN {X 0.121,Y -325.457,Z 632.674,A 0.000,B 0.000,C 90.000,E1 121.209} C_DIS
LIN {X -0.061,Y -336.758,Z 632.658,A 0.000,B 0.000,C 90.000,E1 118.409} C_DIS
LIN {X 0.187,Y -349.487,Z 632.642,A 0.000,B 0.000,C 90.000,E1 115.591} C_DIS
LIN {X -0.010,Y -362.087,Z 632.629,A 0.000,B 0.000,C 90.000,E1 113.206} C_DIS
LIN {X -0.045,Y -375.995,Z 632.616,A 0.000,B 0.000,C 90.000,E1 110.844} C_DIS
LIN {X -0.138,Y -391.308,Z 632.603,A 0.000,B 0.000,C 90.000,E1 108.544} C_DIS
LIN {X 0.037,Y -408.141,Z 632.590,A 0.000,B 0.000,C 90.000,E1 106.260} C_DIS
LIN {X 0.013,Y -426.614,Z 632.578,A 0.000,B 0.000,C 90.000,E1 104.064} C_DIS
LIN {X 0.098,Y -446.499,Z 632.566,A 0.000,B 0.000,C 90.000,E1 101.951} C_DIS
LIN {X 0.123,Y -466.985,Z 632.556,A 0.000,B 0.000,C 90.000,E1 100.018} C_DIS
LIN {X 0.158,Y -472.020,Z 632.553,A 0.000,B 0.000,C 90.000,E1 99.557} C_DIS
LIN {X 0.148,Y -473.946,Z 632.552,A 0.000,B 0.000,C 90.000,E1 99.321} C_DIS
LIN {X 0.061,Y -475.412,Z 632.551,A 0.000,B 0.000,C 90.000,E1 99.095} C_DIS
LIN {X -0.075,Y -476.593,Z 632.549,A 0.000,B 0.000,C 90.000,E1 98.859} C_DIS
LIN {X -0.214,Y -477.452,Z 632.548,A 0.000,B 0.000,C 90.000,E1 98.624} C_DIS
LIN {X -0.075,Y -478.352,Z 632.545,A 0.000,B 0.000,C 90.000,E1 98.106} C_DIS
LIN {X 0.071,Y -478.272,Z 632.542,A 0.000,B 0.000,C 90.000,E1 97.587} C_DIS
LIN {X -0.250,Y -477.203,Z 632.539,A 0.000,B 0.000,C 90.000,E1 97.125} C_DIS
LIN {X 0.092,Y -476.248,Z 632.538,A 0.000,B 0.000,C 90.000,E1 96.834} C_DIS
LIN {X -0.096,Y -474.955,Z 632.537,A 0.000,B 0.000,C 90.000,E1 96.606} C_DIS
LIN {X 0.163,Y -455.894,Z 632.521,A 0.000,B 0.000,C 90.000,E1 93.784} C_DIS
LIN {X 0.085,Y -443.735,Z 632.510,A 0.000,B 0.000,C 90.000,E1 91.718} C_DIS
LIN {X -0.004,Y -433.727,Z 632.499,A 0.000,B 0.000,C 90.000,E1 89.885} C_DIS
LIN {X -0.129,Y -426.245,Z 632.492,A 0.000,B 0.000,C 90.000,E1 88.568} C_DIS
LIN {X -0.114,Y -415.355,Z 632.481,A 0.000,B 0.000,C 90.000,E1 86.674} C_DIS
LIN {X -0.177,Y -401.342,Z 632.468,A 0.000,B 0.000,C 90.000,E1 84.204} C_DIS
LIN {X -0.092,Y -386.421,Z 632.452,A 0.000,B 0.000,C 90.000,E1 81.376} C_DIS
LIN {X 0.094,Y -373.591,Z 632.438,A 0.000,B 0.000,C 90.000,E1 78.757} C_DIS
LIN {X 0.105,Y -362.506,Z 632.425,A 0.000,B 0.000,C 90.000,E1 76.408} C_DIS
LIN {X -0.075,Y -348.153,Z 632.406,A 0.000,B 0.000,C 90.000,E1 73.142} C_DIS
LIN {X 0.038,Y -337.146,Z 632.391,A 0.000,B 0.000,C 90.000,E1 70.369} C_DIS
LIN {X 0.067,Y -323.572,Z 632.370,A 0.000,B 0.000,C 90.000,E1 66.613} C_DIS
LIN {X 0.029,Y -313.434,Z 632.352,A 0.000,B 0.000,C 90.000,E1 63.435} C_DIS
LIN {X -0.034,Y -304.060,Z 632.334,A 0.000,B 0.000,C 90.000,E1 60.205} C_DIS
LIN {X -0.051,Y -295.341,Z 632.316,A 0.000,B 0.000,C 90.000,E1 56.914} C_DIS
LIN {X 0.071,Y -287.141,Z 632.298,A 0.000,B 0.000,C 90.000,E1 53.543} C_DIS
LIN {X -0.062,Y -282.341,Z 632.286,A 0.000,B 0.000,C 90.000,E1 51.537} C_DIS
LIN {X 0.063,Y -277.329,Z 632.275,A 0.000,B 0.000,C 90.000,E1 49.461} C_DIS
LIN {X 0.073,Y -273.748,Z 632.267,A 0.000,B 0.000,C 90.000,E1 48.081} C_DIS
LIN {X 0.037,Y -269.891,Z 632.260,A 0.000,B 0.000,C 90.000,E1 46.701} C_DIS
LIN {X -0.055,Y -265.793,Z 632.252,A 0.000,B 0.000,C 90.000,E1 45.324} C_DIS
LIN {X -0.096,Y -259.214,Z 632.240,A 0.000,B 0.000,C 90.000,E1 43.218} C_DIS
LIN {X -0.051,Y -251.274,Z 632.226,A 0.000,B 0.000,C 90.000,E1 40.701} C_DIS
LIN {X -0.133,Y -241.679,Z 632.208,A 0.000,B 0.000,C 90.000,E1 37.443} C_DIS
LIN {X -0.022,Y -233.815,Z 632.191,A 0.000,B 0.000,C 90.000,E1 34.452} C_DIS
LIN {X -0.117,Y -226.730,Z 632.175,A 0.000,B 0.000,C 90.000,E1 31.465} C_DIS
LIN {X 0.081,Y -220.289,Z 632.158,A 0.000,B 0.000,C 90.000,E1 28.359} C_DIS
LIN {X 0.000,Y -214.631,Z 632.140,A 0.000,B 0.000,C 90.000,E1 25.283} C_DIS
LIN {X 0.026,Y -208.650,Z 632.119,A 0.000,B 0.000,C 90.000,E1 21.354} C_DIS
LIN {X -0.039,Y -203.902,Z 632.097,A 0.000,B 0.000,C 90.000,E1 17.402} C_DIS
LIN {X 0.088,Y -200.143,Z 632.074,A 0.000,B 0.000,C 90.000,E1 13.355} C_DIS
LIN {X 0.053,Y -196.679,Z 632.043,A 0.000,B 0.000,C 90.000,E1 7.701} C_DIS
LIN {X 0.017,Y -197.779,Z 631.952,A 0.000,B 0.000,C 90.000,E1 351.376} C_DIS
LIN {X 0.002,Y -201.228,Z 631.925,A 0.000,B 0.000,C 90.000,E1 346.520} C_DIS
LIN {X 0.042,Y -205.216,Z 631.903,A 0.000,B 0.000,C 90.000,E1 342.489} C_DIS
LIN {X -0.081,Y -210.082,Z 631.881,A 0.000,B 0.000,C 90.000,E1 338.539} C_DIS
LIN {X -0.045,Y -215.769,Z 631.859,A 0.000,B 0.000,C 90.000,E1 334.588} C_DIS
LIN {X 0.068,Y -222.037,Z 631.837,A 0.000,B 0.000,C 90.000,E1 330.667} C_DIS
LIN {X 0.107,Y -227.556,Z 631.820,A 0.000,B 0.000,C 90.000,E1 327.582} C_DIS
LIN {X -0.064,Y -234.941,Z 631.799,A 0.000,B 0.000,C 90.000,E1 323.829} C_DIS
LIN {X 0.028,Y -242.902,Z 631.778,A 0.000,B 0.000,C 90.000,E1 320.070} C_DIS
LIN {X 0.100,Y -251.686,Z 631.758,A 0.000,B 0.000,C 90.000,E1 316.377} C_DIS
LIN {X 0.089,Y -261.493,Z 631.738,A 0.000,B 0.000,C 90.000,E1 312.771} C_DIS
LIN {X -0.175,Y -271.527,Z 631.720,A 0.000,B 0.000,C 90.000,E1 309.644} C_DIS
LIN {X 0.033,Y -284.125,Z 631.701,A 0.000,B 0.000,C 90.000,E1 306.137} C_DIS
LIN {X 0.057,Y -298.298,Z 631.682,A 0.000,B 0.000,C 90.000,E1 302.752} C_DIS
LIN {X 0.062,Y -314.172,Z 631.664,A 0.000,B 0.000,C 90.000,E1 299.461} C_DIS
LIN {X -0.156,Y -329.395,Z 631.648,A 0.000,B 0.000,C 90.000,E1 296.616} C_DIS
LIN {X 0.096,Y -349.093,Z 631.629,A 0.000,B 0.000,C 90.000,E1 293.153} C_DIS
LIN {X 0.099,Y -364.537,Z 631.615,A 0.000,B 0.000,C 90.000,E1 290.737} C_DIS
LIN {X 0.116,Y -379.191,Z 631.604,A 0.000,B 0.000,C 90.000,E1 288.671} C_DIS
LIN {X 0.187,Y -399.769,Z 631.589,A 0.000,B 0.000,C 90.000,E1 286.079} C_DIS
LIN {X -0.081,Y -411.360,Z 631.582,A 0.000,B 0.000,C 90.000,E1 284.717} C_DIS
LIN {X -0.176,Y -422.588,Z 631.574,A 0.000,B 0.000,C 90.000,E1 283.355} C_DIS
LIN {X -0.212,Y -433.357,Z 631.567,A 0.000,B 0.000,C 90.000,E1 282.007} C_DIS
LIN {X -0.083,Y -443.686,Z 631.559,A 0.000,B 0.000,C 90.000,E1 280.658} C_DIS
LIN {X 0.105,Y -457.748,Z 631.549,A 0.000,B 0.000,C 90.000,E1 278.803} C_DIS
LIN {X 0.231,Y -465.617,Z 631.543,A 0.000,B 0.000,C 90.000,E1 277.757} C_DIS
LIN {X 0.137,Y -471.037,Z 631.539,A 0.000,B 0.000,C 90.000,E1 277.004} C_DIS
LIN {X 0.235,Y -474.289,Z 631.536,A 0.000,B 0.000,C 90.000,E1 276.486} C_DIS
LIN {X 0.158,Y -478.343,Z 631.532,A 0.000,B 0.000,C 90.000,E1 275.739} C_DIS
LIN {X -0.175,Y -480.557,Z 631.529,A 0.000,B 0.000,C 90.000,E1 275.277} C_DIS
LIN {X -0.018,Y -482.388,Z 631.526,A 0.000,B 0.000,C 90.000,E1 274.759} C_DIS
LIN {X 0.108,Y -483.811,Z 631.524,A 0.000,B 0.000,C 90.000,E1 274.245} C_DIS
LIN {X -0.201,Y -484.927,Z 631.521,A 0.000,B 0.000,C 90.000,E1 273.784} C_DIS
LIN {X -0.050,Y -485.664,Z 631.518,A 0.000,B 0.000,C 90.000,E1 273.269} C_DIS
LIN {X 0.136,Y -486.093,Z 631.515,A 0.000,B 0.000,C 90.000,E1 272.751} C_DIS
LIN {X -0.184,Y -486.257,Z 631.513,A 0.000,B 0.000,C 90.000,E1 272.293} C_DIS
LIN {X 0.002,Y -486.137,Z 631.510,A 0.000,B 0.000,C 90.000,E1 271.776} C_DIS
LIN {X 0.172,Y -485.653,Z 631.507,A 0.000,B 0.000,C 90.000,E1 271.260} C_DIS
LIN {X -0.142,Y -484.756,Z 631.504,A 0.000,B 0.000,C 90.000,E1 270.802} C_DIS
LIN {X 0.027,Y -483.396,Z 631.502,A 0.000,B 0.000,C 90.000,E1 270.286} C_DIS
LIN {X 0.191,Y -481.451,Z 631.499,A 0.000,B 0.000,C 90.000,E1 269.771} C_DIS
LIN {X -0.135,Y -478.834,Z 631.496,A 0.000,B 0.000,C 90.000,E1 269.312} C_DIS
LIN {X 0.000,Y -475.410,Z 631.493,A 0.000,B 0.000,C 90.000,E1 268.797} C_DIS
LIN {X -0.178,Y -473.365,Z 631.492,A 0.000,B 0.000,C 90.000,E1 268.568} C_DIS
LIN {X -0.057,Y -468.417,Z 631.489,A 0.000,B 0.000,C 90.000,E1 268.051} C_DIS
LIN {X 0.222,Y -465.484,Z 631.488,A 0.000,B 0.000,C 90.000,E1 267.764} C_DIS
LIN {X -0.210,Y -462.451,Z 631.486,A 0.000,B 0.000,C 90.000,E1 267.593} C_DIS
LIN {X -0.178,Y -459.023,Z 631.485,A 0.000,B 0.000,C 90.000,E1 267.364} C_DIS
LIN {X 0.052,Y -451.985,Z 631.483,A 0.000,B 0.000,C 90.000,E1 266.963} C_DIS
LIN {X -0.009,Y -444.517,Z 631.482,A 0.000,B 0.000,C 90.000,E1 266.674} C_DIS
LIN {X -0.012,Y -436.712,Z 631.480,A 0.000,B 0.000,C 90.000,E1 266.445} C_DIS
LIN {X 0.006,Y -428.545,Z 631.479,A 0.000,B 0.000,C 90.000,E1 266.274} C_DIS
LIN {X -0.029,Y -417.640,Z 631.479,A 0.000,B 0.000,C 90.000,E1 266.159} C_DIS
LIN {X -0.160,Y -413.668,Z 631.479,A 0.000,B 0.000,C 90.000,E1 266.159} C_DIS
LIN {X 0.081,Y -180.926,Z 631.479,A 0.000,B 0.000,C 90.000,E1 266.102} C_DIS
LIN {X -0.006,Y -180.899,Z 631.474,A 0.000,B 0.000,C 90.000,E1 265.241} C_DIS
LIN {X -0.056,Y -180.216,Z 631.464,A 0.000,B 0.000,C 90.000,E1 263.571} C_DIS
LIN {X 0.074,Y -179.035,Z 631.445,A 0.000,B 0.000,C 90.000,E1 260.151} C_DIS
LIN {X -0.040,Y -178.694,Z 631.441,A 0.000,B 0.000,C 90.000,E1 259.342} C_DIS
LIN {X 0.071,Y -175.744,Z 631.412,A 0.000,B 0.000,C 90.000,E1 254.212} C_DIS
LIN {X 0.066,Y -171.927,Z 631.384,A 0.000,B 0.000,C 90.000,E1 249.082} C_DIS
LIN {X 0.040,Y -171.302,Z 631.379,A 0.000,B 0.000,C 90.000,E1 248.230} C_DIS
LIN {X 0.086,Y -167.564,Z 631.355,A 0.000,B 0.000,C 90.000,E1 243.896} C_DIS
LIN {X 0.099,Y -166.190,Z 631.345,A 0.000,B 0.000,C 90.000,E1 242.153} C_DIS
LIN {X 0.089,Y -162.959,Z 631.326,A 0.000,B 0.000,C 90.000,E1 238.663} C_DIS
LIN {X -0.087,Y -160.868,Z 631.311,A 0.000,B 0.000,C 90.000,E1 236.087} C_DIS
LIN {X 0.016,Y -157.642,Z 631.292,A 0.000,B 0.000,C 90.000,E1 232.512} C_DIS
LIN {X 0.050,Y -155.679,Z 631.277,A 0.000,B 0.000,C 90.000,E1 229.828} C_DIS
LIN {X -0.005,Y -151.945,Z 631.252,A 0.000,B 0.000,C 90.000,E1 225.364} C_DIS
LIN {X -0.096,Y -150.185,Z 631.237,A 0.000,B 0.000,C 90.000,E1 222.690} C_DIS
LIN {X 0.036,Y -146.957,Z 631.212,A 0.000,B 0.000,C 90.000,E1 218.096} C_DIS
LIN {X -0.061,Y -145.545,Z 631.196,A 0.000,B 0.000,C 90.000,E1 215.391} C_DIS
LIN {X -0.061,Y -142.940,Z 631.171,A 0.000,B 0.000,C 90.000,E1 210.797} C_DIS
LIN {X -0.003,Y -141.564,Z 631.150,A 0.000,B 0.000,C 90.000,E1 207.078} C_DIS
LIN {X 0.049,Y -139.411,Z 631.114,A 0.000,B 0.000,C 90.000,E1 200.556} C_DIS
LIN {X -0.029,Y -139.132,Z 631.104,A 0.000,B 0.000,C 90.000,E1 198.725} C_DIS
LIN {X -0.002,Y -138.349,Z 631.057,A 0.000,B 0.000,C 90.000,E1 190.310} C_DIS
LIN {X -0.015,Y -139.497,Z 631.005,A 0.000,B 0.000,C 90.000,E1 180.974} C_DIS
LIN {X 0.066,Y -141.116,Z 630.974,A 0.000,B 0.000,C 90.000,E1 175.355} C_DIS
LIN {X 0.020,Y -142.496,Z 630.959,A 0.000,B 0.000,C 90.000,E1 172.591} C_DIS
LIN {X -0.034,Y -144.751,Z 630.933,A 0.000,B 0.000,C 90.000,E1 167.993} C_DIS
LIN {X 0.058,Y -147.359,Z 630.913,A 0.000,B 0.000,C 90.000,E1 164.283} C_DIS
LIN {X -0.020,Y -150.685,Z 630.887,A 0.000,B 0.000,C 90.000,E1 159.752} C_DIS
LIN {X 0.063,Y -154.165,Z 630.867,A 0.000,B 0.000,C 90.000,E1 156.102} C_DIS
LIN {X -0.006,Y -157.598,Z 630.847,A 0.000,B 0.000,C 90.000,E1 152.538} C_DIS
LIN {X -0.055,Y -161.848,Z 630.828,A 0.000,B 0.000,C 90.000,E1 148.997} C_DIS
LIN {X -0.037,Y -166.039,Z 630.808,A 0.000,B 0.000,C 90.000,E1 145.468} C_DIS
LIN {X -0.047,Y -171.043,Z 630.789,A 0.000,B 0.000,C 90.000,E1 141.984} C_DIS
LIN {X -0.016,Y -175.913,Z 630.770,A 0.000,B 0.000,C 90.000,E1 138.528} C_DIS
LIN {X -0.024,Y -180.151,Z 630.755,A 0.000,B 0.000,C 90.000,E1 135.972} C_DIS
LIN {X -0.055,Y -185.569,Z 630.737,A 0.000,B 0.000,C 90.000,E1 132.609} C_DIS
LIN {X 0.039,Y -191.097,Z 630.720,A 0.000,B 0.000,C 90.000,E1 129.564} C_DIS
LIN {X 0.007,Y -288.969,Z 630.720,A 0.000,B 0.000,C 90.000,E1 129.564} C_DIS
LIN {X -0.151,Y -290.510,Z 630.720,A 0.000,B 0.000,C 90.000,E1 129.564} C_DIS
LIN {X -0.079,Y -295.557,Z 630.718,A 0.000,B 0.000,C 90.000,E1 129.277} C_DIS
LIN {X 0.101,Y -298.787,Z 630.716,A 0.000,B 0.000,C 90.000,E1 128.910} C_DIS
LIN {X 0.061,Y -302.382,Z 630.713,A 0.000,B 0.000,C 90.000,E1 128.338} C_DIS
LIN {X 0.009,Y -303.818,Z 630.711,A 0.000,B 0.000,C 90.000,E1 128.016} C_DIS
LIN {X 0.010,Y -304.948,Z 630.709,A 0.000,B 0.000,C 90.000,E1 127.684} C_DIS
LIN {X -0.133,Y -315.519,Z 630.689,A 0.000,B 0.000,C 90.000,E1 124.119} C_DIS
LIN {X 0.013,Y -325.506,Z 630.673,A 0.000,B 0.000,C 90.000,E1 121.209} C_DIS
LIN {X 0.125,Y -336.816,Z 630.658,A 0.000,B 0.000,C 90.000,E1 118.359} C_DIS
LIN {X 0.075,Y -349.554,Z 630.642,A 0.000,B 0.000,C 90.000,E1 115.591} C_DIS
LIN {X -0.124,Y -362.165,Z 630.629,A 0.000,B 0.000,C 90.000,E1 113.206} C_DIS
LIN {X 0.190,Y -376.082,Z 630.616,A 0.000,B 0.000,C 90.000,E1 110.791} C_DIS
LIN {X 0.114,Y -391.406,Z 630.603,A 0.000,B 0.000,C 90.000,E1 108.489} C_DIS
LIN {X -0.084,Y -408.250,Z 630.590,A 0.000,B 0.000,C 90.000,E1 106.260} C_DIS
LIN {X -0.112,Y -426.736,Z 630.578,A 0.000,B 0.000,C 90.000,E1 104.064} C_DIS
LIN {X -0.024,Y -446.628,Z 630.566,A 0.000,B 0.000,C 90.000,E1 101.951} C_DIS
LIN {X 0.004,Y -467.119,Z 630.556,A 0.000,B 0.000,C 90.000,E1 100.018} C_DIS
LIN {X 0.041,Y -472.146,Z 630.553,A 0.000,B 0.000,C 90.000,E1 99.557} C_DIS
LIN {X 0.027,Y -474.067,Z 630.552,A 0.000,B 0.000,C 90.000,E1 99.321} C_DIS
LIN {X -0.063,Y -475.530,Z 630.550,A 0.000,B 0.000,C 90.000,E1 99.095} C_DIS
LIN {X 0.134,Y -477.559,Z 630.548,A 0.000,B 0.000,C 90.000,E1 98.568} C_DIS
LIN {X -0.205,Y -478.452,Z 630.545,A 0.000,B 0.000,C 90.000,E1 98.106} C_DIS
LIN {X -0.059,Y -478.363,Z 630.542,A 0.000,B 0.000,C 90.000,E1 97.587} C_DIS
LIN {X 0.095,Y -477.284,Z 630.539,A 0.000,B 0.000,C 90.000,E1 97.068} C_DIS
LIN {X -0.037,Y -476.324,Z 630.538,A 0.000,B 0.000,C 90.000,E1 96.834} C_DIS
LIN {X -0.224,Y -475.023,Z 630.537,A 0.000,B 0.000,C 90.000,E1 96.606} C_DIS
LIN {X -0.187,Y -457.574,Z 630.522,A 0.000,B 0.000,C 90.000,E1 94.069} C_DIS
LIN {X 0.005,Y -446.682,Z 630.512,A 0.000,B 0.000,C 90.000,E1 92.236} C_DIS
LIN {X 0.154,Y -435.190,Z 630.501,A 0.000,B 0.000,C 90.000,E1 90.115} C_DIS
LIN {X 0.051,Y -427.780,Z 630.493,A 0.000,B 0.000,C 90.000,E1 88.797} C_DIS
LIN {X -0.036,Y -418.500,Z 630.484,A 0.000,B 0.000,C 90.000,E1 87.192} C_DIS
LIN {X -0.185,Y -407.505,Z 630.474,A 0.000,B 0.000,C 90.000,E1 85.298} C_DIS
LIN {X 0.018,Y -393.814,Z 630.460,A 0.000,B 0.000,C 90.000,E1 82.761} C_DIS
LIN {X -0.071,Y -379.253,Z 630.444,A 0.000,B 0.000,C 90.000,E1 79.926} C_DIS
LIN {X -0.015,Y -366.676,Z 630.429,A 0.000,B 0.000,C 90.000,E1 77.297} C_DIS
LIN {X -0.058,Y -351.980,Z 630.411,A 0.000,B 0.000,C 90.000,E1 74.031} C_DIS
LIN {X 0.064,Y -339.606,Z 630.394,A 0.000,B 0.000,C 90.000,E1 70.967} C_DIS
LIN {X 0.069,Y -325.807,Z 630.374,A 0.000,B 0.000,C 90.000,E1 67.230} C_DIS
LIN {X -0.038,Y -313.550,Z 630.352,A 0.000,B 0.000,C 90.000,E1 63.435} C_DIS
LIN {X -0.096,Y -304.184,Z 630.334,A 0.000,B 0.000,C 90.000,E1 60.205} C_DIS
LIN {X -0.107,Y -295.452,Z 630.316,A 0.000,B 0.000,C 90.000,E1 56.914} C_DIS
LIN {X 0.019,Y -287.244,Z 630.297,A 0.000,B 0.000,C 90.000,E1 53.543} C_DIS
LIN {X -0.111,Y -282.445,Z 630.286,A 0.000,B 0.000,C 90.000,E1 51.537} C_DIS
LIN {X 0.018,Y -277.441,Z 630.275,A 0.000,B 0.000,C 90.000,E1 49.461} C_DIS
LIN {X 0.019,Y -271.947,Z 630.263,A 0.000,B 0.000,C 90.000,E1 47.391} C_DIS
LIN {X -0.095,Y -265.898,Z 630.252,A 0.000,B 0.000,C 90.000,E1 45.324} C_DIS
LIN {X 0.055,Y -259.289,Z 630.240,A 0.000,B 0.000,C 90.000,E1 43.176} C_DIS
LIN {X -0.068,Y -250.234,Z 630.224,A 0.000,B 0.000,C 90.000,E1 40.334} C_DIS
LIN {X 0.010,Y -239.712,Z 630.204,A 0.000,B 0.000,C 90.000,E1 36.664} C_DIS
LIN {X -0.064,Y -232.039,Z 630.187,A 0.000,B 0.000,C 90.000,E1 33.706} C_DIS
LIN {X -0.006,Y -225.141,Z 630.170,A 0.000,B 0.000,C 90.000,E1 30.669} C_DIS
LIN {X 0.044,Y -218.857,Z 630.153,A 0.000,B 0.000,C 90.000,E1 27.590} C_DIS
LIN {X -0.071,Y -213.421,Z 630.136,A 0.000,B 0.000,C 90.000,E1 24.515} C_DIS
LIN {X 0.029,Y -207.660,Z 630.114,A 0.000,B 0.000,C 90.000,E1 20.556} C_DIS
LIN {X 0.064,Y -203.126,Z 630.092,A 0.000,B 0.000,C 90.000,E1 16.567} C_DIS
LIN {X -0.076,Y -199.588,Z 630.070,A 0.000,B 0.000,C 90.000,E1 12.591} C_DIS
LIN {X 0.027,Y -196.410,Z 630.038,A 0.000,B 0.000,C 90.000,E1 6.891} C_DIS
LIN {X 0.031,Y -197.391,Z 629.957,A 0.000,B 0.000,C 90.000,E1 352.186} C_DIS
LIN {X -0.082,Y -200.601,Z 629.930,A 0.000,B 0.000,C 90.000,E1 347.353} C_DIS
LIN {X -0.067,Y -204.407,Z 629.907,A 0.000,B 0.000,C 90.000,E1 343.323} C_DIS
LIN {X -0.086,Y -209.080,Z 629.885,A 0.000,B 0.000,C 90.000,E1 339.337} C_DIS
LIN {X 0.026,Y -214.634,Z 629.863,A 0.000,B 0.000,C 90.000,E1 335.357} C_DIS
LIN {X 0.000,Y -220.764,Z 629.841,A 0.000,B 0.000,C 90.000,E1 331.463} C_DIS
LIN {X 0.122,Y -227.570,Z 629.820,A 0.000,B 0.000,C 90.000,E1 327.582} C_DIS
LIN {X -0.048,Y -234.964,Z 629.799,A 0.000,B 0.000,C 90.000,E1 323.829} C_DIS
LIN {X 0.045,Y -242.911,Z 629.778,A 0.000,B 0.000,C 90.000,E1 320.070} C_DIS
LIN {X 0.118,Y -251.656,Z 629.758,A 0.000,B 0.000,C 90.000,E1 316.377} C_DIS
LIN {X 0.106,Y -261.446,Z 629.738,A 0.000,B 0.000,C 90.000,E1 312.771} C_DIS
LIN {X -0.028,Y -270.258,Z 629.722,A 0.000,B 0.000,C 90.000,E1 309.967} C_DIS
LIN {X -0.072,Y -282.709,Z 629.703,A 0.000,B 0.000,C 90.000,E1 306.503} C_DIS
LIN {X 0.067,Y -296.729,Z 629.684,A 0.000,B 0.000,C 90.000,E1 303.086} C_DIS
LIN {X 0.020,Y -312.388,Z 629.666,A 0.000,B 0.000,C 90.000,E1 299.795} C_DIS
LIN {X 0.106,Y -325.822,Z 629.651,A 0.000,B 0.000,C 90.000,E1 297.206} C_DIS
LIN {X 0.074,Y -343.450,Z 629.634,A 0.000,B 0.000,C 90.000,E1 294.079} C_DIS
LIN {X 0.035,Y -362.452,Z 629.617,A 0.000,B 0.000,C 90.000,E1 291.046} C_DIS
LIN {X 0.116,Y -379.155,Z 629.604,A 0.000,B 0.000,C 90.000,E1 288.671} C_DIS
LIN {X 0.186,Y -399.721,Z 629.589,A 0.000,B 0.000,C 90.000,E1 286.079} C_DIS
LIN {X 0.028,Y -413.597,Z 629.580,A 0.000,B 0.000,C 90.000,E1 284.426} C_DIS
LIN {X -0.037,Y -424.730,Z 629.573,A 0.000,B 0.000,C 90.000,E1 283.063} C_DIS
LIN {X -0.030,Y -435.417,Z 629.565,A 0.000,B 0.000,C 90.000,E1 281.715} C_DIS
LIN {X 0.129,Y -445.698,Z 629.558,A 0.000,B 0.000,C 90.000,E1 280.366} C_DIS
LIN {X -0.083,Y -459.646,Z 629.548,A 0.000,B 0.000,C 90.000,E1 278.568} C_DIS
LIN {X -0.004,Y -467.320,Z 629.542,A 0.000,B 0.000,C 90.000,E1 277.530} C_DIS
LIN {X -0.088,Y -472.583,Z 629.538,A 0.000,B 0.000,C 90.000,E1 276.777} C_DIS
LIN {X 0.020,Y -475.603,Z 629.535,A 0.000,B 0.000,C 90.000,E1 276.258} C_DIS
LIN {X -0.041,Y -479.356,Z 629.531,A 0.000,B 0.000,C 90.000,E1 275.511} C_DIS
LIN {X -0.184,Y -480.447,Z 629.529,A 0.000,B 0.000,C 90.000,E1 275.277} C_DIS
LIN {X -0.029,Y -482.299,Z 629.526,A 0.000,B 0.000,C 90.000,E1 274.759} C_DIS
LIN {X 0.097,Y -483.718,Z 629.524,A 0.000,B 0.000,C 90.000,E1 274.245} C_DIS
LIN {X -0.213,Y -484.862,Z 629.521,A 0.000,B 0.000,C 90.000,E1 273.784} C_DIS
LIN {X -0.062,Y -485.614,Z 629.518,A 0.000,B 0.000,C 90.000,E1 273.269} C_DIS
LIN {X 0.123,Y -486.075,Z 629.515,A 0.000,B 0.000,C 90.000,E1 272.751} C_DIS
LIN {X -0.197,Y -486.225,Z 629.513,A 0.000,B 0.000,C 90.000,E1 272.293} C_DIS
LIN {X -0.011,Y -486.104,Z 629.510,A 0.000,B 0.000,C 90.000,E1 271.776} C_DIS
LIN {X 0.159,Y -485.653,Z 629.507,A 0.000,B 0.000,C 90.000,E1 271.260} C_DIS
LIN {X -0.155,Y -484.743,Z 629.504,A 0.000,B 0.000,C 90.000,E1 270.802} C_DIS
LIN {X 0.014,Y -483.377,Z 629.502,A 0.000,B 0.000,C 90.000,E1 270.286} C_DIS
LIN {X 0.177,Y -481.445,Z 629.499,A 0.000,B 0.000,C 90.000,E1 269.771} C_DIS
LIN {X -0.148,Y -478.866,Z 629.496,A 0.000,B 0.000,C 90.000,E1 269.312} C_DIS
LIN {X -0.013,Y -475.436,Z 629.493,A 0.000,B 0.000,C 90.000,E1 268.797} C_DIS
LIN {X 0.102,Y -471.084,Z 629.491,A 0.000,B 0.000,C 90.000,E1 268.282} C_DIS
LIN {X 0.209,Y -465.506,Z 629.488,A 0.000,B 0.000,C 90.000,E1 267.764} C_DIS
LIN {X -0.223,Y -458.994,Z 629.485,A 0.000,B 0.000,C 90.000,E1 267.364} C_DIS
LIN {X -0.026,Y -451.861,Z 629.483,A 0.000,B 0.000,C 90.000,E1 266.963} C_DIS
LIN {X -0.093,Y -444.206,Z 629.481,A 0.000,B 0.000,C 90.000,E1 266.674} C_DIS
LIN {X -0.047,Y -436.624,Z 629.480,A 0.000,B 0.000,C 90.000,E1 266.445} C_DIS
LIN {X -0.059,Y -428.054,Z 629.479,A 0.000,B 0.000,C 90.000,E1 266.274} C_DIS
LIN {X -0.080,Y -416.907,Z 629.479,A 0.000,B 0.000,C 90.000,E1 266.159} C_DIS
LIN {X -0.209,Y -413.008,Z 629.479,A 0.000,B 0.000,C 90.000,E1 266.159} C_DIS
LIN {X 0.060,Y -180.925,Z 629.478,A 0.000,B 0.000,C 90.000,E1 266.102} C_DIS
LIN {X -0.025,Y -180.899,Z 629.474,A 0.000,B 0.000,C 90.000,E1 265.241} C_DIS
LIN {X -0.075,Y -180.214,Z 629.464,A 0.000,B 0.000,C 90.000,E1 263.571} C_DIS
LIN {X 0.055,Y -179.033,Z 629.445,A 0.000,B 0.000,C 90.000,E1 260.151} C_DIS
LIN {X -0.059,Y -178.690,Z 629.441,A 0.000,B 0.000,C 90.000,E1 259.342} C_DIS
LIN {X 0.052,Y -175.740,Z 629.412,A 0.000,B 0.000,C 90.000,E1 254.212} C_DIS
LIN {X 0.048,Y -171.923,Z 629.384,A 0.000,B 0.000,C 90.000,E1 249.082} C_DIS
LIN {X 0.022,Y -171.296,Z 629.379,A 0.000,B 0.000,C 90.000,E1 248.230} C_DIS
LIN {X 0.068,Y -167.559,Z 629.355,A 0.000,B 0.000,C 90.000,E1 243.896} C_DIS
LIN {X 0.081,Y -166.184,Z 629.345,A 0.000,B 0.000,C 90.000,E1 242.153} C_DIS
LIN {X 0.070,Y -162.954,Z 629.326,A 0.000,B 0.000,C 90.000,E1 238.663} C_DIS
LIN {X -0.106,Y -160.862,Z 629.311,A 0.000,B 0.000,C 90.000,E1 236.087} C_DIS
LIN {X 0.095,Y -157.637,Z 629.292,A 0.000,B 0.000,C 90.000,E1 232.477} C_DIS
LIN {X 0.032,Y -155.674,Z 629.277,A 0.000,B 0.000,C 90.000,E1 229.828} C_DIS
LIN {X 0.084,Y -151.941,Z 629.252,A 0.000,B 0.000,C 90.000,E1 225.324} C_DIS
LIN {X 0.099,Y -150.179,Z 629.237,A 0.000,B 0.000,C 90.000,E1 222.609} C_DIS
LIN {X 0.018,Y -146.954,Z 629.212,A 0.000,B 0.000,C 90.000,E1 218.096} C_DIS
LIN {X 0.006,Y -145.541,Z 629.196,A 0.000,B 0.000,C 90.000,E1 215.358} C_DIS
LIN {X -0.078,Y -142.937,Z 629.171,A 0.000,B 0.000,C 90.000,E1 210.797} C_DIS
LIN {X -0.020,Y -141.562,Z 629.150,A 0.000,B 0.000,C 90.000,E1 207.078} C_DIS
LIN {X 0.032,Y -139.409,Z 629.114,A 0.000,B 0.000,C 90.000,E1 200.556} C_DIS
LIN {X -0.046,Y -139.130,Z 629.104,A 0.000,B 0.000,C 90.000,E1 198.725} C_DIS
LIN {X -0.018,Y -138.351,Z 629.057,A 0.000,B 0.000,C 90.000,E1 190.310} C_DIS
LIN {X -0.031,Y -139.498,Z 629.005,A 0.000,B 0.000,C 90.000,E1 180.974} C_DIS
LIN {X 0.050,Y -141.119,Z 628.974,A 0.000,B 0.000,C 90.000,E1 175.355} C_DIS
LIN {X 0.003,Y -142.499,Z 628.959,A 0.000,B 0.000,C 90.000,E1 172.591} C_DIS
LIN {X -0.050,Y -144.754,Z 628.933,A 0.000,B 0.000,C 90.000,E1 167.993} C_DIS
LIN {X 0.041,Y -147.364,Z 628.913,A 0.000,B 0.000,C 90.000,E1 164.283} C_DIS
LIN {X -0.037,Y -150.690,Z 628.887,A 0.000,B 0.000,C 90.000,E1 159.752} C_DIS
LIN {X 0.046,Y -154.171,Z 628.867,A 0.000,B 0.000,C 90.000,E1 156.102} C_DIS
LIN {X -0.024,Y -157.605,Z 628.847,A 0.000,B 0.000,C 90.000,E1 152.538} C_DIS
LIN {X -0.074,Y -161.857,Z 628.828,A 0.000,B 0.000,C 90.000,E1 148.997} C_DIS
LIN {X -0.056,Y -166.048,Z 628.808,A 0.000,B 0.000,C 90.000,E1 145.468} C_DIS
LIN {X -0.065,Y -171.052,Z 628.789,A 0.000,B 0.000,C 90.000,E1 141.984} C_DIS
LIN {X -0.035,Y -175.923,Z 628.770,A 0.000,B 0.000,C 90.000,E1 138.528} C_DIS
LIN {X -0.042,Y -180.162,Z 628.755,A 0.000,B 0.000,C 90.000,E1 135.972} C_DIS
LIN {X -0.074,Y -185.579,Z 628.737,A 0.000,B 0.000,C 90.000,E1 132.609} C_DIS
LIN {X 0.020,Y -191.106,Z 628.720,A 0.000,B 0.000,C 90.000,E1 129.564} C_DIS
LIN {X -0.023,Y -289.001,Z 628.720,A 0.000,B 0.000,C 90.000,E1 129.564} C_DIS
LIN {X 0.042,Y -290.522,Z 628.720,A 0.000,B 0.000,C 90.000,E1 129.519} C_DIS
LIN {X -0.110,Y -295.556,Z 628.718,A 0.000,B 0.000,C 90.000,E1 129.277} C_DIS
LIN {X 0.066,Y -298.790,Z 628.716,A 0.000,B 0.000,C 90.000,E1 128.910} C_DIS
LIN {X 0.023,Y -302.384,Z 628.713,A 0.000,B 0.000,C 90.000,E1 128.338} C_DIS
LIN {X -0.028,Y -303.819,Z 628.711,A 0.000,B 0.000,C 90.000,E1 128.016} C_DIS
LIN {X -0.027,Y -304.947,Z 628.709,A 0.000,B 0.000,C 90.000,E1 127.684} C_DIS
LIN {X 0.089,Y -315.521,Z 628.689,A 0.000,B 0.000,C 90.000,E1 124.072} C_DIS
LIN {X -0.028,Y -325.512,Z 628.673,A 0.000,B 0.000,C 90.000,E1 121.209} C_DIS
LIN {X 0.083,Y -336.824,Z 628.658,A 0.000,B 0.000,C 90.000,E1 118.359} C_DIS
LIN {X 0.033,Y -349.566,Z 628.642,A 0.000,B 0.000,C 90.000,E1 115.591} C_DIS
LIN {X -0.168,Y -362.180,Z 628.629,A 0.000,B 0.000,C 90.000,E1 113.206} C_DIS
LIN {X 0.144,Y -376.101,Z 628.616,A 0.000,B 0.000,C 90.000,E1 110.791} C_DIS
LIN {X 0.067,Y -391.429,Z 628.603,A 0.000,B 0.000,C 90.000,E1 108.489} C_DIS
LIN {X -0.133,Y -408.277,Z 628.590,A 0.000,B 0.000,C 90.000,E1 106.260} C_DIS
LIN {X -0.162,Y -426.768,Z 628.578,A 0.000,B 0.000,C 90.000,E1 104.064} C_DIS
LIN {X -0.074,Y -446.663,Z 628.566,A 0.000,B 0.000,C 90.000,E1 101.951} C_DIS
LIN {X -0.044,Y -467.155,Z 628.556,A 0.000,B 0.000,C 90.000,E1 100.018} C_DIS
LIN {X -0.007,Y -472.195,Z 628.553,A 0.000,B 0.000,C 90.000,E1 99.557} C_DIS
LIN {X -0.015,Y -474.123,Z 628.552,A 0.000,B 0.000,C 90.000,E1 99.321} C_DIS
LIN {X -0.099,Y -475.592,Z 628.550,A 0.000,B 0.000,C 90.000,E1 99.095} C_DIS
LIN {X -0.236,Y -476.776,Z 628.549,A 0.000,B 0.000,C 90.000,E1 98.859} C_DIS
LIN {X 0.097,Y -477.639,Z 628.548,A 0.000,B 0.000,C 90.000,E1 98.568} C_DIS
LIN {X -0.235,Y -478.545,Z 628.545,A 0.000,B 0.000,C 90.000,E1 98.106} C_DIS
LIN {X -0.087,Y -478.470,Z 628.542,A 0.000,B 0.000,C 90.000,E1 97.587} C_DIS
LIN {X 0.067,Y -477.405,Z 628.539,A 0.000,B 0.000,C 90.000,E1 97.068} C_DIS
LIN {X -0.065,Y -476.454,Z 628.538,A 0.000,B 0.000,C 90.000,E1 96.834} C_DIS
LIN {X -0.251,Y -475.165,Z 628.537,A 0.000,B 0.000,C 90.000,E1 96.606} C_DIS
LIN {X 0.019,Y -456.051,Z 628.521,A 0.000,B 0.000,C 90.000,E1 93.784} C_DIS
LIN {X -0.051,Y -443.865,Z 628.510,A 0.000,B 0.000,C 90.000,E1 91.718} C_DIS
LIN {X -0.133,Y -433.841,Z 628.499,A 0.000,B 0.000,C 90.000,E1 89.885} C_DIS
LIN {X 0.171,Y -426.348,Z 628.492,A 0.000,B 0.000,C 90.000,E1 88.511} C_DIS
LIN {X 0.054,Y -417.007,Z 628.483,A 0.000,B 0.000,C 90.000,E1 86.906} C_DIS
LIN {X 0.061,Y -402.965,Z 628.469,A 0.000,B 0.000,C 90.000,E1 84.432} C_DIS
LIN {X 0.139,Y -389.467,Z 628.455,A 0.000,B 0.000,C 90.000,E1 81.894} C_DIS
LIN {X -0.020,Y -375.096,Z 628.439,A 0.000,B 0.000,C 90.000,E1 79.050} C_DIS
LIN {X 0.030,Y -363.999,Z 628.426,A 0.000,B 0.000,C 90.000,E1 76.700} C_DIS
LIN {X -0.090,Y -349.538,Z 628.408,A 0.000,B 0.000,C 90.000,E1 73.433} C_DIS
LIN {X -0.044,Y -338.503,Z 628.393,A 0.000,B 0.000,C 90.000,E1 70.678} C_DIS
LIN {X 0.075,Y -325.922,Z 628.374,A 0.000,B 0.000,C 90.000,E1 67.230} C_DIS
LIN {X -0.028,Y -313.687,Z 628.352,A 0.000,B 0.000,C 90.000,E1 63.435} C_DIS
LIN {X -0.081,Y -304.327,Z 628.334,A 0.000,B 0.000,C 90.000,E1 60.205} C_DIS
LIN {X -0.088,Y -295.600,Z 628.316,A 0.000,B 0.000,C 90.000,E1 56.914} C_DIS
LIN {X 0.042,Y -287.382,Z 628.297,A 0.000,B 0.000,C 90.000,E1 53.543} C_DIS
LIN {X -0.086,Y -282.581,Z 628.286,A 0.000,B 0.000,C 90.000,E1 51.537} C_DIS
LIN {X 0.044,Y -277.555,Z 628.275,A 0.000,B 0.000,C 90.000,E1 49.461} C_DIS
LIN {X 0.057,Y -273.968,Z 628.267,A 0.000,B 0.000,C 90.000,E1 48.081} C_DIS
LIN {X 0.025,Y -270.115,Z 628.259,A 0.000,B 0.000,C 90.000,E1 46.701} C_DIS
LIN {X -0.065,Y -266.020,Z 628.252,A 0.000,B 0.000,C 90.000,E1 45.324} C_DIS
LIN {X 0.088,Y -259.418,Z 628.240,A 0.000,B 0.000,C 90.000,E1 43.176} C_DIS
LIN {X -0.033,Y -250.353,Z 628.224,A 0.000,B 0.000,C 90.000,E1 40.334} C_DIS
LIN {X 0.046,Y -239.812,Z 628.204,A 0.000,B 0.000,C 90.000,E1 36.664} C_DIS
LIN {X -0.027,Y -232.155,Z 628.187,A 0.000,B 0.000,C 90.000,E1 33.706} C_DIS
LIN {X 0.033,Y -225.246,Z 628.170,A 0.000,B 0.000,C 90.000,E1 30.669} C_DIS
LIN {X 0.084,Y -218.951,Z 628.153,A 0.000,B 0.000,C 90.000,E1 27.590} C_DIS
LIN {X -0.030,Y -213.509,Z 628.136,A 0.000,B 0.000,C 90.000,E1 24.515} C_DIS
LIN {X 0.045,Y -208.800,Z 628.119,A 0.000,B 0.000,C 90.000,E1 21.354} C_DIS
LIN {X -0.017,Y -204.027,Z 628.097,A 0.000,B 0.000,C 90.000,E1 17.402} C_DIS
LIN {X -0.080,Y -200.277,Z 628.074,A 0.000,B 0.000,C 90.000,E1 13.411} C_DIS
LIN {X 0.089,Y -197.141,Z 628.047,A 0.000,B 0.000,C 90.000,E1 8.511} C_DIS
LIN {X 0.024,Y -197.882,Z 627.952,A 0.000,B 0.000,C 90.000,E1 351.376} C_DIS
LIN {X 0.013,Y -201.331,Z 627.925,A 0.000,B 0.000,C 90.000,E1 346.520} C_DIS
LIN {X 0.057,Y -205.342,Z 627.903,A 0.000,B 0.000,C 90.000,E1 342.489} C_DIS
LIN {X -0.061,Y -210.196,Z 627.881,A 0.000,B 0.000,C 90.000,E1 338.539} C_DIS
LIN {X -0.021,Y -215.836,Z 627.859,A 0.000,B 0.000,C 90.000,E1 334.588} C_DIS
LIN {X 0.095,Y -222.096,Z 627.837,A 0.000,B 0.000,C 90.000,E1 330.667} C_DIS
LIN {X 0.137,Y -227.593,Z 627.820,A 0.000,B 0.000,C 90.000,E1 327.582} C_DIS
LIN {X -0.034,Y -234.985,Z 627.799,A 0.000,B 0.000,C 90.000,E1 323.829} C_DIS
LIN {X 0.062,Y -242.921,Z 627.778,A 0.000,B 0.000,C 90.000,E1 320.070} C_DIS
LIN {X 0.135,Y -251.639,Z 627.758,A 0.000,B 0.000,C 90.000,E1 316.377} C_DIS
LIN {X 0.123,Y -261.400,Z 627.738,A 0.000,B 0.000,C 90.000,E1 312.771} C_DIS
LIN {X -0.012,Y -270.175,Z 627.722,A 0.000,B 0.000,C 90.000,E1 309.967} C_DIS
LIN {X -0.057,Y -282.632,Z 627.703,A 0.000,B 0.000,C 90.000,E1 306.503} C_DIS
LIN {X 0.080,Y -296.632,Z 627.684,A 0.000,B 0.000,C 90.000,E1 303.086} C_DIS
LIN {X 0.030,Y -312.273,Z 627.666,A 0.000,B 0.000,C 90.000,E1 299.795} C_DIS
LIN {X 0.113,Y -325.721,Z 627.651,A 0.000,B 0.000,C 90.000,E1 297.206} C_DIS
LIN {X 0.077,Y -343.348,Z 627.634,A 0.000,B 0.000,C 90.000,E1 294.079} C_DIS
LIN {X -0.017,Y -360.380,Z 627.619,A 0.000,B 0.000,C 90.000,E1 291.354} C_DIS
LIN {X 0.115,Y -379.092,Z 627.604,A 0.000,B 0.000,C 90.000,E1 288.671} C_DIS
LIN {X 0.184,Y -399.694,Z 627.589,A 0.000,B 0.000,C 90.000,E1 286.079} C_DIS
LIN {X 0.025,Y -413.565,Z 627.580,A 0.000,B 0.000,C 90.000,E1 284.426} C_DIS
LIN {X -0.041,Y -424.689,Z 627.573,A 0.000,B 0.000,C 90.000,E1 283.063} C_DIS
LIN {X -0.035,Y -435.401,Z 627.565,A 0.000,B 0.000,C 90.000,E1 281.715} C_DIS
LIN {X 0.123,Y -445.688,Z 627.558,A 0.000,B 0.000,C 90.000,E1 280.366} C_DIS
LIN {X 0.095,Y -457.622,Z 627.549,A 0.000,B 0.000,C 90.000,E1 278.803} C_DIS
LIN {X -0.011,Y -467.196,Z 627.542,A 0.000,B 0.000,C 90.000,E1 277.530} C_DIS
LIN {X -0.097,Y -472.441,Z 627.538,A 0.000,B 0.000,C 90.000,E1 276.777} C_DIS
LIN {X -0.137,Y -476.805,Z 627.533,A 0.000,B 0.000,C 90.000,E1 276.024} C_DIS
LIN {X -0.195,Y -480.335,Z 627.529,A 0.000,B 0.000,C 90.000,E1 275.277} C_DIS
LIN {X -0.040,Y -482.203,Z 627.526,A 0.000,B 0.000,C 90.000,E1 274.759} C_DIS
LIN {X 0.085,Y -483.671,Z 627.524,A 0.000,B 0.000,C 90.000,E1 274.245} C_DIS
LIN {X -0.225,Y -484.783,Z 627.521,A 0.000,B 0.000,C 90.000,E1 273.784} C_DIS
LIN {X -0.075,Y -485.567,Z 627.518,A 0.000,B 0.000,C 90.000,E1 273.269} C_DIS
LIN {X 0.110,Y -486.047,Z 627.515,A 0.000,B 0.000,C 90.000,E1 272.751} C_DIS
LIN {X -0.211,Y -486.215,Z 627.513,A 0.000,B 0.000,C 90.000,E1 272.293} C_DIS
LIN {X -0.024,Y -486.094,Z 627.510,A 0.000,B 0.000,C 90.000,E1 271.776} C_DIS
LIN {X 0.146,Y -485.629,Z 627.507,A 0.000,B 0.000,C 90.000,E1 271.260} C_DIS
LIN {X -0.169,Y -484.750,Z 627.504,A 0.000,B 0.000,C 90.000,E1 270.802} C_DIS
LIN {X 0.000,Y -483.385,Z 627.502,A 0.000,B 0.000,C 90.000,E1 270.286} C_DIS
LIN {X 0.164,Y -481.480,Z 627.499,A 0.000,B 0.000,C 90.000,E1 269.771} C_DIS
LIN {X -0.162,Y -478.907,Z 627.496,A 0.000,B 0.000,C 90.000,E1 269.312} C_DIS
LIN {X -0.026,Y -475.466,Z 627.493,A 0.000,B 0.000,C 90.000,E1 268.797} C_DIS
LIN {X 0.090,Y -471.076,Z 627.491,A 0.000,B 0.000,C 90.000,E1 268.282} C_DIS
LIN {X -0.084,Y -468.454,Z 627.489,A 0.000,B 0.000,C 90.000,E1 268.051} C_DIS
LIN {X 0.197,Y -465.501,Z 627.488,A 0.000,B 0.000,C 90.000,E1 267.764} C_DIS
LIN {X -0.186,Y -459.076,Z 627.485,A 0.000,B 0.000,C 90.000,E1 267.364} C_DIS
LIN {X 0.152,Y -455.845,Z 627.484,A 0.000,B 0.000,C 90.000,E1 267.135} C_DIS
LIN {X -0.191,Y -448.644,Z 627.482,A 0.000,B 0.000,C 90.000,E1 266.846} C_DIS
LIN {X 0.023,Y -441.170,Z 627.481,A 0.000,B 0.000,C 90.000,E1 266.560} C_DIS
LIN {X -0.197,Y -433.265,Z 627.480,A 0.000,B 0.000,C 90.000,E1 266.388} C_DIS
LIN {X -0.016,Y -424.107,Z 627.479,A 0.000,B 0.000,C 90.000,E1 266.216} C_DIS
LIN {X -0.173,Y -414.564,Z 627.479,A 0.000,B 0.000,C 90.000,E1 266.159} C_DIS
LIN {X 0.169,Y -412.291,Z 627.478,A 0.000,B 0.000,C 90.000,E1 266.102} C_DIS
LIN {X 0.044,Y -180.926,Z 627.478,A 0.000,B 0.000,C 90.000,E1 266.102} C_DIS
LIN {X -0.020,Y -180.899,Z 627.474,A 0.000,B 0.000,C 90.000,E1 265.241} C_DIS
LIN {X -0.070,Y -180.215,Z 627.464,A 0.000,B 0.000,C 90.000,E1 263.571} C_DIS
LIN {X 0.060,Y -179.034,Z 627.445,A 0.000,B 0.000,C 90.000,E1 260.151} C_DIS
LIN {X -0.054,Y -178.691,Z 627.441,A 0.000,B 0.000,C 90.000,E1 259.342} C_DIS
LIN {X 0.057,Y -175.740,Z 627.412,A 0.000,B 0.000,C 90.000,E1 254.212} C_DIS
LIN {X 0.052,Y -171.924,Z 627.384,A 0.000,B 0.000,C 90.000,E1 249.082} C_DIS
LIN {X 0.027,Y -171.297,Z 627.379,A 0.000,B 0.000,C 90.000,E1 248.230} C_DIS
LIN {X 0.072,Y -167.561,Z 627.355,A 0.000,B 0.000,C 90.000,E1 243.896} C_DIS
LIN {X 0.086,Y -166.186,Z 627.345,A 0.000,B 0.000,C 90.000,E1 242.153} C_DIS
LIN {X 0.075,Y -162.956,Z 627.326,A 0.000,B 0.000,C 90.000,E1 238.663} C_DIS
LIN {X -0.101,Y -160.864,Z 627.311,A 0.000,B 0.000,C 90.000,E1 236.087} C_DIS
LIN {X 0.099,Y -157.638,Z 627.292,A 0.000,B 0.000,C 90.000,E1 232.477} C_DIS
LIN {X 0.037,Y -155.675,Z 627.277,A 0.000,B 0.000,C 90.000,E1 229.828} C_DIS
LIN {X -0.018,Y -151.943,Z 627.252,A 0.000,B 0.000,C 90.000,E1 225.364} C_DIS
LIN {X 0.104,Y -150.180,Z 627.237,A 0.000,B 0.000,C 90.000,E1 222.609} C_DIS
LIN {X 0.022,Y -146.955,Z 627.212,A 0.000,B 0.000,C 90.000,E1 218.096} C_DIS
LIN {X 0.010,Y -145.542,Z 627.196,A 0.000,B 0.000,C 90.000,E1 215.358} C_DIS
LIN {X -0.073,Y -142.937,Z 627.171,A 0.000,B 0.000,C 90.000,E1 210.797} C_DIS
LIN {X -0.015,Y -141.562,Z 627.150,A 0.000,B 0.000,C 90.000,E1 207.078} C_DIS
LIN {X 0.037,Y -139.409,Z 627.114,A 0.000,B 0.000,C 90.000,E1 200.556} C_DIS
LIN {X -0.042,Y -139.131,Z 627.104,A 0.000,B 0.000,C 90.000,E1 198.725} C_DIS
LIN {X -0.014,Y -138.350,Z 627.057,A 0.000,B 0.000,C 90.000,E1 190.310} C_DIS
LIN {X -0.027,Y -139.498,Z 627.005,A 0.000,B 0.000,C 90.000,E1 180.974} C_DIS
LIN {X 0.055,Y -141.119,Z 626.974,A 0.000,B 0.000,C 90.000,E1 175.355} C_DIS
LIN {X 0.008,Y -142.499,Z 626.959,A 0.000,B 0.000,C 90.000,E1 172.591} C_DIS
LIN {X -0.046,Y -144.753,Z 626.933,A 0.000,B 0.000,C 90.000,E1 167.993} C_DIS
LIN {X 0.046,Y -147.362,Z 626.913,A 0.000,B 0.000,C 90.000,E1 164.283} C_DIS
LIN {X -0.033,Y -150.689,Z 626.887,A 0.000,B 0.000,C 90.000,E1 159.752} C_DIS
LIN {X 0.050,Y -154.170,Z 626.867,A 0.000,B 0.000,C 90.000,E1 156.102} C_DIS
LIN {X -0.019,Y -157.603,Z 626.847,A 0.000,B 0.000,C 90.000,E1 152.538} C_DIS
LIN {X -0.069,Y -161.855,Z 626.828,A 0.000,B 0.000,C 90.000,E1 148.997} C_DIS
LIN {X -0.052,Y -166.045,Z 626.808,A 0.000,B 0.000,C 90.000,E1 145.468} C_DIS
LIN {X -0.060,Y -171.050,Z 626.789,A 0.000,B 0.000,C 90.000,E1 141.984} C_DIS
LIN {X -0.030,Y -175.920,Z 626.770,A 0.000,B 0.000,C 90.000,E1 138.528} C_DIS
LIN {X -0.037,Y -180.159,Z 626.755,A 0.000,B 0.000,C 90.000,E1 135.972} C_DIS
LIN {X -0.069,Y -185.576,Z 626.737,A 0.000,B 0.000,C 90.000,E1 132.609} C_DIS
LIN {X -0.012,Y -191.121,Z 626.720,A 0.000,B 0.000,C 90.000,E1 129.564} C_DIS
LIN {X -0.070,Y -289.045,Z 626.720,A 0.000,B 0.000,C 90.000,E1 129.564} C_DIS
LIN {X 0.048,Y -290.149,Z 626.720,A 0.000,B 0.000,C 90.000,E1 129.519} C_DIS
LIN {X -0.102,Y -295.433,Z 626.718,A 0.000,B 0.000,C 90.000,E1 129.277} C_DIS
LIN {X -0.080,Y -298.590,Z 626.716,A 0.000,B 0.000,C 90.000,E1 128.955} C_DIS
LIN {X -0.073,Y -302.213,Z 626.713,A 0.000,B 0.000,C 90.000,E1 128.382} C_DIS
LIN {X 0.114,Y -303.685,Z 626.711,A 0.000,B 0.000,C 90.000,E1 128.016} C_DIS
LIN {X -0.128,Y -304.843,Z 626.709,A 0.000,B 0.000,C 90.000,E1 127.729} C_DIS
LIN {X -0.029,Y -315.417,Z 626.690,A 0.000,B 0.000,C 90.000,E1 124.119} C_DIS
LIN {X 0.116,Y -325.396,Z 626.674,A 0.000,B 0.000,C 90.000,E1 121.209} C_DIS
LIN {X -0.068,Y -336.697,Z 626.658,A 0.000,B 0.000,C 90.000,E1 118.409} C_DIS
LIN {X 0.180,Y -349.424,Z 626.642,A 0.000,B 0.000,C 90.000,E1 115.591} C_DIS
LIN {X -0.019,Y -362.026,Z 626.629,A 0.000,B 0.000,C 90.000,E1 113.206} C_DIS
LIN {X -0.056,Y -375.932,Z 626.616,A 0.000,B 0.000,C 90.000,E1 110.844} C_DIS
LIN {X -0.152,Y -391.247,Z 626.603,A 0.000,B 0.000,C 90.000,E1 108.544} C_DIS
LIN {X 0.022,Y -408.079,Z 626.590,A 0.000,B 0.000,C 90.000,E1 106.260} C_DIS
LIN {X -0.005,Y -426.554,Z 626.578,A 0.000,B 0.000,C 90.000,E1 104.064} C_DIS
LIN {X 0.077,Y -446.439,Z 626.566,A 0.000,B 0.000,C 90.000,E1 101.951} C_DIS
LIN {X 0.100,Y -466.926,Z 626.556,A 0.000,B 0.000,C 90.000,E1 100.018} C_DIS
LIN {X 0.135,Y -472.020,Z 626.553,A 0.000,B 0.000,C 90.000,E1 99.557} C_DIS
LIN {X 0.154,Y -473.993,Z 626.552,A 0.000,B 0.000,C 90.000,E1 99.321} C_DIS
LIN {X 0.096,Y -475.498,Z 626.551,A 0.000,B 0.000,C 90.000,E1 99.095} C_DIS
LIN {X -0.040,Y -476.733,Z 626.549,A 0.000,B 0.000,C 90.000,E1 98.859} C_DIS
LIN {X -0.178,Y -477.637,Z 626.548,A 0.000,B 0.000,C 90.000,E1 98.624} C_DIS
LIN {X -0.039,Y -478.614,Z 626.545,A 0.000,B 0.000,C 90.000,E1 98.106} C_DIS
LIN {X 0.109,Y -478.607,Z 626.542,A 0.000,B 0.000,C 90.000,E1 97.587} C_DIS
LIN {X -0.211,Y -477.615,Z 626.539,A 0.000,B 0.000,C 90.000,E1 97.125} C_DIS
LIN {X -0.056,Y -475.467,Z 626.537,A 0.000,B 0.000,C 90.000,E1 96.606} C_DIS
LIN {X -0.055,Y -470.187,Z 626.532,A 0.000,B 0.000,C 90.000,E1 95.853} C_DIS
LIN {X 0.223,Y -456.346,Z 626.521,A 0.000,B 0.000,C 90.000,E1 93.784} C_DIS
LIN {X -0.099,Y -442.677,Z 626.508,A 0.000,B 0.000,C 90.000,E1 91.489} C_DIS
LIN {X -0.206,Y -432.633,Z 626.498,A 0.000,B 0.000,C 90.000,E1 89.656} C_DIS
LIN {X 0.084,Y -425.085,Z 626.491,A 0.000,B 0.000,C 90.000,E1 88.282} C_DIS
LIN {X -0.030,Y -415.689,Z 626.482,A 0.000,B 0.000,C 90.000,E1 86.674} C_DIS
LIN {X 0.001,Y -400.183,Z 626.466,A 0.000,B 0.000,C 90.000,E1 83.913} C_DIS
LIN {X 0.004,Y -386.773,Z 626.452,A 0.000,B 0.000,C 90.000,E1 81.376} C_DIS
LIN {X -0.170,Y -373.919,Z 626.438,A 0.000,B 0.000,C 90.000,E1 78.814} C_DIS
LIN {X -0.169,Y -361.513,Z 626.423,A 0.000,B 0.000,C 90.000,E1 76.172} C_DIS
LIN {X -0.035,Y -347.266,Z 626.405,A 0.000,B 0.000,C 90.000,E1 72.851} C_DIS
LIN {X 0.159,Y -337.521,Z 626.391,A 0.000,B 0.000,C 90.000,E1 70.369} C_DIS
LIN {X -0.094,Y -324.027,Z 626.370,A 0.000,B 0.000,C 90.000,E1 66.666} C_DIS
LIN {X 0.035,Y -313.933,Z 626.353,A 0.000,B 0.000,C 90.000,E1 63.461} C_DIS
LIN {X 0.124,Y -304.574,Z 626.335,A 0.000,B 0.000,C 90.000,E1 60.205} C_DIS
LIN {X 0.118,Y -295.819,Z 626.316,A 0.000,B 0.000,C 90.000,E1 56.914} C_DIS
LIN {X 0.079,Y -287.598,Z 626.298,A 0.000,B 0.000,C 90.000,E1 53.577} C_DIS
LIN {X 0.123,Y -282.790,Z 626.286,A 0.000,B 0.000,C 90.000,E1 51.537} C_DIS
LIN {X -0.139,Y -277.786,Z 626.275,A 0.000,B 0.000,C 90.000,E1 49.542} C_DIS
LIN {X -0.129,Y -272.304,Z 626.264,A 0.000,B 0.000,C 90.000,E1 47.472} C_DIS
LIN {X 0.004,Y -268.343,Z 626.256,A 0.000,B 0.000,C 90.000,E1 46.053} C_DIS
LIN {X 0.009,Y -261.901,Z 626.244,A 0.000,B 0.000,C 90.000,E1 43.947} C_DIS
LIN {X -0.077,Y -253.946,Z 626.230,A 0.000,B 0.000,C 90.000,E1 41.472} C_DIS
LIN {X 0.060,Y -244.131,Z 626.212,A 0.000,B 0.000,C 90.000,E1 38.177} C_DIS
LIN {X 0.038,Y -236.080,Z 626.196,A 0.000,B 0.000,C 90.000,E1 35.231} C_DIS
LIN {X -0.070,Y -228.806,Z 626.179,A 0.000,B 0.000,C 90.000,E1 32.260} C_DIS
LIN {X -0.014,Y -220.622,Z 626.158,A 0.000,B 0.000,C 90.000,E1 28.437} C_DIS
LIN {X 0.013,Y -214.936,Z 626.141,A 0.000,B 0.000,C 90.000,E1 25.335} C_DIS
LIN {X 0.043,Y -208.936,Z 626.119,A 0.000,B 0.000,C 90.000,E1 21.408} C_DIS
LIN {X -0.020,Y -204.131,Z 626.097,A 0.000,B 0.000,C 90.000,E1 17.457} C_DIS
LIN {X 0.112,Y -200.376,Z 626.075,A 0.000,B 0.000,C 90.000,E1 13.411} C_DIS
LIN {X 0.086,Y -197.212,Z 626.048,A 0.000,B 0.000,C 90.000,E1 8.568} C_DIS
LIN {X 0.028,Y -197.934,Z 625.952,A 0.000,B 0.000,C 90.000,E1 351.376} C_DIS
LIN {X 0.019,Y -201.382,Z 625.925,A 0.000,B 0.000,C 90.000,E1 346.520} C_DIS
LIN {X 0.065,Y -205.402,Z 625.903,A 0.000,B 0.000,C 90.000,E1 342.489} C_DIS
LIN {X -0.051,Y -210.252,Z 625.881,A 0.000,B 0.000,C 90.000,E1 338.539} C_DIS
LIN {X -0.008,Y -215.869,Z 625.859,A 0.000,B 0.000,C 90.000,E1 334.588} C_DIS
LIN {X -0.086,Y -222.125,Z 625.837,A 0.000,B 0.000,C 90.000,E1 330.717} C_DIS
LIN {X 0.029,Y -227.614,Z 625.820,A 0.000,B 0.000,C 90.000,E1 327.612} C_DIS
LIN {X -0.017,Y -235.008,Z 625.799,A 0.000,B 0.000,C 90.000,E1 323.829} C_DIS
LIN {X 0.078,Y -242.924,Z 625.778,A 0.000,B 0.000,C 90.000,E1 320.070} C_DIS
LIN {X -0.029,Y -251.617,Z 625.758,A 0.000,B 0.000,C 90.000,E1 316.419} C_DIS
LIN {X 0.140,Y -261.343,Z 625.738,A 0.000,B 0.000,C 90.000,E1 312.771} C_DIS
LIN {X 0.004,Y -270.091,Z 625.722,A 0.000,B 0.000,C 90.000,E1 309.967} C_DIS
LIN {X -0.044,Y -282.546,Z 625.703,A 0.000,B 0.000,C 90.000,E1 306.503} C_DIS
LIN {X 0.092,Y -296.535,Z 625.684,A 0.000,B 0.000,C 90.000,E1 303.086} C_DIS
LIN {X 0.040,Y -312.159,Z 625.666,A 0.000,B 0.000,C 90.000,E1 299.795} C_DIS
LIN {X -0.079,Y -327.355,Z 625.649,A 0.000,B 0.000,C 90.000,E1 296.924} C_DIS
LIN {X 0.089,Y -346.924,Z 625.630,A 0.000,B 0.000,C 90.000,E1 293.462} C_DIS
LIN {X -0.016,Y -360.301,Z 625.619,A 0.000,B 0.000,C 90.000,E1 291.354} C_DIS
LIN {X 0.113,Y -379.028,Z 625.604,A 0.000,B 0.000,C 90.000,E1 288.671} C_DIS
LIN {X 0.182,Y -399.633,Z 625.589,A 0.000,B 0.000,C 90.000,E1 286.079} C_DIS
LIN {X 0.021,Y -413.532,Z 625.580,A 0.000,B 0.000,C 90.000,E1 284.426} C_DIS
LIN {X -0.045,Y -424.663,Z 625.573,A 0.000,B 0.000,C 90.000,E1 283.063} C_DIS
LIN {X -0.040,Y -435.385,Z 625.565,A 0.000,B 0.000,C 90.000,E1 281.715} C_DIS
LIN {X 0.118,Y -445.686,Z 625.558,A 0.000,B 0.000,C 90.000,E1 280.366} C_DIS
LIN {X 0.090,Y -457.552,Z 625.549,A 0.000,B 0.000,C 90.000,E1 278.803} C_DIS
LIN {X -0.018,Y -467.087,Z 625.542,A 0.000,B 0.000,C 90.000,E1 277.530} C_DIS
LIN {X -0.104,Y -472.316,Z 625.538,A 0.000,B 0.000,C 90.000,E1 276.777} C_DIS
LIN {X -0.146,Y -476.679,Z 625.533,A 0.000,B 0.000,C 90.000,E1 276.024} C_DIS
LIN {X -0.205,Y -480.231,Z 625.529,A 0.000,B 0.000,C 90.000,E1 275.277} C_DIS
LIN {X -0.050,Y -482.096,Z 625.526,A 0.000,B 0.000,C 90.000,E1 274.759} C_DIS
LIN {X 0.074,Y -483.613,Z 625.524,A 0.000,B 0.000,C 90.000,E1 274.245} C_DIS
LIN {X -0.237,Y -484.742,Z 625.521,A 0.000,B 0.000,C 90.000,E1 273.784} C_DIS
LIN {X -0.087,Y -485.502,Z 625.518,A 0.000,B 0.000,C 90.000,E1 273.269} C_DIS
LIN {X 0.098,Y -485.999,Z 625.515,A 0.000,B 0.000,C 90.000,E1 272.751} C_DIS
LIN {X -0.223,Y -486.229,Z 625.513,A 0.000,B 0.000,C 90.000,E1 272.293} C_DIS
LIN {X -0.038,Y -486.091,Z 625.510,A 0.000,B 0.000,C 90.000,E1 271.776} C_DIS
LIN {X 0.133,Y -485.595,Z 625.507,A 0.000,B 0.000,C 90.000,E1 271.260} C_DIS
LIN {X -0.182,Y -484.738,Z 625.504,A 0.000,B 0.000,C 90.000,E1 270.802} C_DIS
LIN {X -0.013,Y -483.394,Z 625.502,A 0.000,B 0.000,C 90.000,E1 270.286} C_DIS
LIN {X 0.150,Y -481.507,Z 625.499,A 0.000,B 0.000,C 90.000,E1 269.771} C_DIS
LIN {X -0.175,Y -478.898,Z 625.496,A 0.000,B 0.000,C 90.000,E1 269.312} C_DIS
LIN {X 0.132,Y -477.328,Z 625.495,A 0.000,B 0.000,C 90.000,E1 269.026} C_DIS
LIN {X -0.217,Y -473.416,Z 625.492,A 0.000,B 0.000,C 90.000,E1 268.568} C_DIS
LIN {X 0.077,Y -471.135,Z 625.490,A 0.000,B 0.000,C 90.000,E1 268.282} C_DIS
LIN {X -0.096,Y -468.492,Z 625.489,A 0.000,B 0.000,C 90.000,E1 268.051} C_DIS
LIN {X 0.184,Y -465.526,Z 625.488,A 0.000,B 0.000,C 90.000,E1 267.764} C_DIS
LIN {X -0.188,Y -459.211,Z 625.485,A 0.000,B 0.000,C 90.000,E1 267.364} C_DIS
LIN {X 0.137,Y -455.882,Z 625.484,A 0.000,B 0.000,C 90.000,E1 267.135} C_DIS
LIN {X 0.232,Y -448.562,Z 625.482,A 0.000,B 0.000,C 90.000,E1 266.788} C_DIS
LIN {X -0.011,Y -441.094,Z 625.481,A 0.000,B 0.000,C 90.000,E1 266.560} C_DIS
LIN {X 0.200,Y -433.056,Z 625.480,A 0.000,B 0.000,C 90.000,E1 266.331} C_DIS
